Yaskawa INFORM job: DEMO_ROOF_UPPER_0625_3PAINT_66.JBI

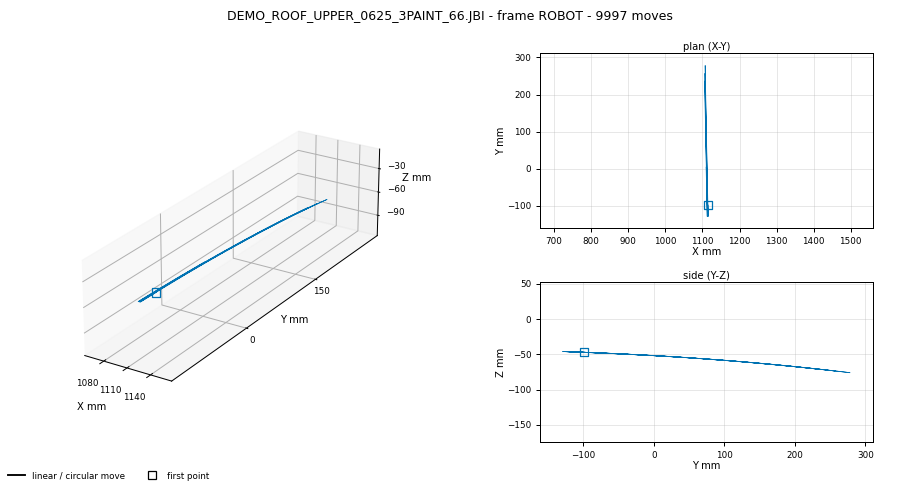
[picture p0: tool path of DEMO_ROOF_UPPER_0625_3PAINT_66.JBI in frame ROBOT, 9997 of 9997 moves have a stored position in this frame; points joined in program order, loops and branches not executed]
/JOB
//NAME DEMO_ROOF_UPPER_0625_3PAINT66
//POS
///NPOS 9997,0,0,0,0,0
///TOOL 0
///USER 0
///POSTYPE ROBOT
///RECTAN
///RCONF 1,0,0,0,0,0,0,0,0,0,0,0,0,0,0,0,0,0,0,0,0,0,0,0
C00000=1115.021,-98.188,-46.924,179.727,4.538,148.836
C00001=1115.026,-98.438,-46.914,179.727,4.533,148.835
C00002=1115.031,-98.688,-46.905,179.727,4.528,148.834
C00003=1115.036,-98.938,-46.894,179.727,4.523,148.833
C00004=1115.041,-99.188,-46.885,179.728,4.519,148.832
C00005=1115.047,-99.437,-46.875,179.728,4.513,148.830
C00006=1115.052,-99.653,-46.868,179.729,4.509,148.829
C00007=1115.056,-99.868,-46.859,179.728,4.505,148.828
C00008=1115.061,-100.083,-46.851,179.729,4.500,148.827
C00009=1115.066,-100.298,-46.842,179.729,4.496,148.826
C00010=1115.070,-100.513,-46.834,179.730,4.492,148.825
C00011=1115.075,-100.728,-46.826,179.729,4.488,148.824
C00012=1115.079,-100.943,-46.819,179.730,4.483,148.823
C00013=1115.084,-101.159,-46.811,179.731,4.479,148.822
C00014=1115.089,-101.408,-46.800,179.731,4.474,148.821
C00015=1115.094,-101.658,-46.791,179.731,4.469,148.820
C00016=1115.100,-101.908,-46.781,179.731,4.464,148.819
C00017=1115.105,-102.158,-46.772,179.732,4.459,148.817
C00018=1115.110,-102.407,-46.763,179.732,4.454,148.816
C00019=1115.116,-102.657,-46.753,179.733,4.449,148.815
C00020=1115.121,-102.907,-46.744,179.733,4.444,148.814
C00021=1115.127,-103.156,-46.734,179.733,4.439,148.813
C00022=1115.132,-103.406,-46.725,179.733,4.434,148.812
C00023=1115.137,-103.656,-46.716,179.734,4.429,148.810
C00024=1115.143,-103.906,-46.706,179.734,4.424,148.809
C00025=1115.148,-104.155,-46.697,179.735,4.419,148.808
C00026=1115.153,-104.405,-46.688,179.735,4.414,148.807
C00027=1115.159,-104.655,-46.678,179.735,4.409,148.806
C00028=1115.164,-104.905,-46.669,179.735,4.404,148.804
C00029=1115.170,-105.155,-46.660,179.736,4.399,148.803
C00030=1115.174,-105.404,-46.650,179.736,4.394,148.802
C00031=1115.180,-105.654,-46.641,179.737,4.389,148.801
C00032=1115.186,-105.904,-46.632,179.737,4.384,148.800
C00033=1115.190,-106.153,-46.622,179.737,4.379,148.798
C00034=1115.196,-106.403,-46.613,179.737,4.373,148.797
C00035=1115.201,-106.653,-46.604,179.738,4.369,148.796
C00036=1115.207,-106.903,-46.595,179.738,4.364,148.795
C00037=1115.211,-107.152,-46.585,179.739,4.359,148.794
C00038=1115.217,-107.402,-46.576,179.739,4.354,148.792
C00039=1115.223,-107.652,-46.567,179.739,4.348,148.791
C00040=1115.228,-107.902,-46.558,179.739,4.343,148.790
C00041=1115.233,-108.151,-46.548,179.739,4.338,148.789
C00042=1115.238,-108.402,-46.539,179.740,4.333,148.788
C00043=1115.244,-108.651,-46.530,179.741,4.329,148.786
C00044=1115.249,-108.901,-46.521,179.741,4.323,148.785
C00045=1115.254,-109.151,-46.512,179.741,4.318,148.784
C00046=1115.260,-109.401,-46.502,179.741,4.313,148.783
C00047=1115.265,-109.651,-46.493,179.742,4.308,148.782
C00048=1115.270,-109.900,-46.484,179.742,4.303,148.780
C00049=1115.275,-110.150,-46.475,179.742,4.298,148.779
C00050=1115.282,-110.400,-46.466,179.742,4.292,148.778
C00051=1115.287,-110.650,-46.457,179.743,4.287,148.777
C00052=1115.292,-110.899,-46.448,179.743,4.282,148.776
C00053=1115.297,-111.149,-46.439,179.743,4.277,148.774
C00054=1115.302,-111.399,-46.430,179.743,4.272,148.773
C00055=1115.308,-111.649,-46.420,179.744,4.267,148.772
C00056=1115.313,-111.899,-46.411,179.744,4.262,148.771
C00057=1115.318,-112.148,-46.402,179.745,4.257,148.770
C00058=1115.323,-112.398,-46.394,179.745,4.252,148.768
C00059=1115.329,-112.648,-46.385,179.745,4.247,148.767
C00060=1115.335,-112.898,-46.376,179.745,4.242,148.766
C00061=1115.340,-113.147,-46.367,179.746,4.236,148.764
C00062=1115.344,-113.363,-46.359,179.746,4.231,148.763
C00063=1115.349,-113.578,-46.350,179.746,4.227,148.763
C00064=1115.354,-113.793,-46.343,179.747,4.223,148.761
C00065=1115.359,-114.008,-46.335,179.747,4.218,148.760
C00066=1115.363,-114.223,-46.327,179.747,4.214,148.759
C00067=1115.367,-114.438,-46.320,179.747,4.209,148.758
C00068=1115.372,-114.654,-46.312,179.748,4.205,148.757
C00069=1115.376,-114.869,-46.305,179.748,4.200,148.756
C00070=1115.382,-115.118,-46.296,179.748,4.195,148.755
C00071=1115.388,-115.369,-46.286,179.749,4.190,148.754
C00072=1115.393,-115.619,-46.278,179.749,4.184,148.752
C00073=1115.398,-115.868,-46.269,179.749,4.179,148.751
C00074=1115.404,-116.118,-46.260,179.749,4.174,148.750
C00075=1115.409,-116.367,-46.251,179.750,4.169,148.749
C00076=1115.414,-116.617,-46.242,179.750,4.164,148.748
C00077=1115.419,-116.867,-46.233,179.751,4.158,148.746
C00078=1115.424,-117.117,-46.225,179.751,4.153,148.745
C00079=1115.430,-117.366,-46.216,179.751,4.148,148.744
C00080=1115.435,-117.616,-46.207,179.752,4.143,148.742
C00081=1115.441,-117.867,-46.198,179.752,4.137,148.741
C00082=1115.447,-118.117,-46.189,179.752,4.132,148.740
C00083=1115.452,-118.366,-46.181,179.752,4.127,148.739
C00084=1115.458,-118.616,-46.172,179.753,4.122,148.737
C00085=1115.463,-118.865,-46.163,179.753,4.116,148.736
C00086=1115.468,-119.115,-46.154,179.754,4.111,148.735
C00087=1115.473,-119.365,-46.145,179.754,4.106,148.734
C00088=1115.479,-119.614,-46.137,179.754,4.101,148.733
C00089=1115.484,-119.865,-46.129,179.755,4.096,148.731
C00090=1115.489,-120.115,-46.120,179.755,4.090,148.730
C00091=1115.495,-120.364,-46.111,179.755,4.084,148.729
C00092=1115.500,-120.614,-46.102,179.755,4.079,148.727
C00093=1115.506,-120.863,-46.093,179.756,4.074,148.726
C00094=1115.511,-121.113,-46.085,179.756,4.069,148.725
C00095=1115.516,-121.364,-46.076,179.757,4.063,148.724
C00096=1115.522,-121.613,-46.068,179.757,4.058,148.722
C00097=1115.527,-121.863,-46.059,179.757,4.053,148.721
C00098=1115.532,-122.113,-46.050,179.758,4.048,148.720
C00099=1115.538,-122.363,-46.042,179.758,4.042,148.718
C00100=1115.544,-122.612,-46.033,179.758,4.036,148.717
C00101=1115.549,-122.862,-46.024,179.758,4.031,148.716
C00102=1115.553,-123.112,-46.016,179.759,4.026,148.715
C00103=1115.559,-123.362,-46.008,179.760,4.020,148.713
C00104=1115.564,-123.611,-45.999,179.760,4.015,148.712
C00105=1115.570,-123.861,-45.990,179.760,4.010,148.711
C00106=1115.575,-124.111,-45.982,179.760,4.005,148.710
C00107=1115.581,-124.361,-45.974,179.761,3.998,148.708
C00108=1115.586,-124.611,-45.965,179.761,3.993,148.707
C00109=1115.591,-124.860,-45.956,179.761,3.988,148.706
C00110=1115.597,-125.110,-45.948,179.762,3.983,148.705
C00111=1115.602,-125.360,-45.939,179.762,3.977,148.703
C00112=1115.607,-125.610,-45.930,179.762,3.971,148.702
C00113=1115.613,-125.859,-45.923,179.762,3.966,148.701
C00114=1115.618,-126.109,-45.914,179.763,3.961,148.699
C00115=1115.623,-126.360,-45.906,179.763,3.955,148.698
C00116=1115.629,-126.609,-45.898,179.764,3.950,148.697
C00117=1115.634,-126.859,-45.889,179.764,3.944,148.695
C00118=1115.640,-127.074,-45.882,179.764,3.940,148.694
C00119=1115.644,-127.289,-45.875,179.765,3.935,148.693
C00120=1115.648,-127.504,-45.867,179.765,3.930,148.692
C00121=1115.654,-127.720,-45.860,179.765,3.926,148.691
C00122=1115.658,-127.935,-45.853,179.766,3.920,148.690
C00123=1115.662,-128.151,-45.845,179.765,3.916,148.689
C00124=1115.667,-128.366,-45.838,179.766,3.911,148.688
C00125=1115.671,-128.581,-45.831,179.767,3.906,148.686
C00126=1115.248,-128.571,-45.857,179.774,3.911,148.685
C00127=1115.243,-128.356,-45.864,179.774,3.916,148.686
C00128=1115.239,-128.141,-45.872,179.773,3.920,148.687
C00129=1115.234,-127.926,-45.878,179.773,3.925,148.689
C00130=1115.229,-127.710,-45.886,179.773,3.929,148.689
C00131=1115.225,-127.496,-45.893,179.772,3.934,148.691
C00132=1115.221,-127.280,-45.901,179.772,3.939,148.692
C00133=1115.216,-127.064,-45.908,179.772,3.943,148.693
C00134=1115.212,-126.849,-45.915,179.771,3.949,148.694
C00135=1115.206,-126.600,-45.923,179.771,3.954,148.695
C00136=1115.201,-126.350,-45.932,179.770,3.959,148.697
C00137=1115.195,-126.100,-45.941,179.770,3.965,148.698
C00138=1115.190,-125.851,-45.949,179.770,3.970,148.699
C00139=1115.184,-125.600,-45.957,179.769,3.976,148.701
C00140=1115.179,-125.350,-45.966,179.769,3.981,148.702
C00141=1115.173,-125.101,-45.975,179.769,3.986,148.703
C00142=1115.168,-124.851,-45.982,179.768,3.993,148.705
C00143=1115.163,-124.601,-45.991,179.768,3.998,148.706
C00144=1115.158,-124.351,-46.000,179.768,4.003,148.707
C00145=1115.152,-124.102,-46.008,179.768,4.008,148.708
C00146=1115.147,-123.852,-46.017,179.767,4.014,148.710
C00147=1115.142,-123.602,-46.026,179.766,4.019,148.711
C00148=1115.136,-123.353,-46.034,179.767,4.025,148.712
C00149=1115.130,-123.102,-46.042,179.766,4.030,148.713
C00150=1115.125,-122.853,-46.051,179.766,4.036,148.715
C00151=1115.120,-122.603,-46.060,179.765,4.041,148.716
C00152=1115.114,-122.354,-46.069,179.765,4.046,148.717
C00153=1115.109,-122.104,-46.078,179.765,4.051,148.718
C00154=1115.104,-121.853,-46.086,179.764,4.057,148.720
C00155=1115.099,-121.603,-46.095,179.764,4.062,148.721
C00156=1115.093,-121.354,-46.103,179.764,4.068,148.722
C00157=1115.088,-121.104,-46.112,179.764,4.073,148.724
C00158=1115.082,-120.854,-46.121,179.763,4.079,148.725
C00159=1115.077,-120.604,-46.129,179.763,4.084,148.726
C00160=1115.071,-120.355,-46.138,179.762,4.089,148.727
C00161=1115.066,-120.105,-46.147,179.762,4.094,148.729
C00162=1115.061,-119.855,-46.156,179.762,4.099,148.730
C00163=1115.056,-119.605,-46.164,179.761,4.105,148.731
C00164=1115.051,-119.355,-46.173,179.761,4.110,148.733
C00165=1115.045,-119.106,-46.182,179.760,4.115,148.734
C00166=1115.040,-118.856,-46.191,179.760,4.120,148.735
C00167=1115.034,-118.607,-46.200,179.760,4.125,148.736
C00168=1115.029,-118.356,-46.208,179.760,4.131,148.737
C00169=1115.024,-118.106,-46.217,179.759,4.136,148.739
C00170=1115.018,-117.857,-46.225,179.758,4.141,148.740
C00171=1115.013,-117.607,-46.234,179.759,4.147,148.741
C00172=1115.007,-117.357,-46.244,179.758,4.152,148.742
C00173=1115.002,-117.107,-46.253,179.758,4.158,148.744
C00174=1114.997,-116.857,-46.261,179.758,4.163,148.745
C00175=1114.991,-116.608,-46.270,179.757,4.168,148.746
C00176=1114.986,-116.358,-46.279,179.757,4.173,148.748
C00177=1114.981,-116.109,-46.288,179.757,4.179,148.749
C00178=1114.975,-115.859,-46.297,179.756,4.184,148.750
C00179=1114.970,-115.609,-46.306,179.756,4.189,148.751
C00180=1114.965,-115.359,-46.314,179.756,4.194,148.752
C00181=1114.959,-115.109,-46.324,179.756,4.199,148.754
C00182=1114.953,-114.860,-46.333,179.755,4.204,148.755
C00183=1114.949,-114.644,-46.340,179.754,4.209,148.756
C00184=1114.944,-114.429,-46.348,179.755,4.214,148.757
C00185=1114.940,-114.214,-46.356,179.754,4.218,148.758
C00186=1114.935,-113.999,-46.363,179.754,4.222,148.759
C00187=1114.931,-113.784,-46.371,179.754,4.227,148.760
C00188=1114.927,-113.569,-46.379,179.753,4.231,148.761
C00189=1114.922,-113.354,-46.387,179.753,4.236,148.762
C00190=1114.917,-113.138,-46.394,179.753,4.240,148.763
C00191=1114.911,-112.888,-46.404,179.752,4.245,148.765
C00192=1114.906,-112.638,-46.413,179.752,4.251,148.766
C00193=1114.901,-112.389,-46.422,179.752,4.256,148.767
C00194=1114.896,-112.139,-46.430,179.751,4.261,148.768
C00195=1114.891,-111.889,-46.439,179.751,4.266,148.769
C00196=1114.885,-111.639,-46.450,179.751,4.271,148.771
C00197=1114.879,-111.390,-46.458,179.751,4.276,148.772
C00198=1114.874,-111.140,-46.467,179.750,4.282,148.773
C00199=1114.869,-110.891,-46.476,179.749,4.286,148.774
C00200=1114.863,-110.640,-46.485,179.749,4.291,148.776
C00201=1114.858,-110.391,-46.494,179.749,4.296,148.777
C00202=1114.853,-110.141,-46.504,179.749,4.301,148.778
C00203=1114.848,-109.891,-46.513,179.748,4.307,148.779
C00204=1114.842,-109.641,-46.522,179.748,4.312,148.780
C00205=1114.837,-109.391,-46.531,179.748,4.317,148.782
C00206=1114.831,-109.142,-46.540,179.748,4.322,148.783
C00207=1114.827,-108.892,-46.550,179.747,4.327,148.784
C00208=1114.821,-108.642,-46.559,179.747,4.332,148.785
C00209=1114.816,-108.392,-46.568,179.746,4.337,148.786
C00210=1114.810,-108.142,-46.577,179.746,4.342,148.788
C00211=1114.804,-107.892,-46.586,179.746,4.347,148.789
C00212=1114.800,-107.643,-46.596,179.746,4.352,148.790
C00213=1114.794,-107.393,-46.605,179.745,4.357,148.791
C00214=1114.789,-107.143,-46.614,179.745,4.362,148.792
C00215=1114.784,-106.894,-46.624,179.745,4.368,148.794
C00216=1114.779,-106.644,-46.633,179.745,4.373,148.795
C00217=1114.773,-106.394,-46.642,179.743,4.378,148.796
C00218=1114.767,-106.144,-46.651,179.743,4.383,148.797
C00219=1114.763,-105.895,-46.661,179.743,4.388,148.799
C00220=1114.757,-105.645,-46.670,179.743,4.393,148.800
C00221=1114.752,-105.395,-46.679,179.742,4.398,148.801
C00222=1114.747,-105.145,-46.689,179.743,4.403,148.802
C00223=1114.741,-104.895,-46.698,179.742,4.408,148.803
C00224=1114.736,-104.645,-46.707,179.742,4.412,148.804
C00225=1114.731,-104.396,-46.717,179.741,4.418,148.805
C00226=1114.725,-104.146,-46.727,179.741,4.423,148.807
C00227=1114.720,-103.896,-46.735,179.741,4.428,148.808
C00228=1114.715,-103.647,-46.745,179.741,4.433,148.809
C00229=1114.709,-103.397,-46.755,179.740,4.437,148.810
C00230=1114.704,-103.148,-46.764,179.740,4.443,148.811
C00231=1114.698,-102.897,-46.774,179.739,4.448,148.813
C00232=1114.693,-102.648,-46.783,179.739,4.453,148.814
C00233=1114.688,-102.398,-46.792,179.739,4.458,148.815
C00234=1114.682,-102.148,-46.802,179.739,4.463,148.816
C00235=1114.677,-101.899,-46.811,179.738,4.468,148.817
C00236=1114.671,-101.649,-46.821,179.738,4.473,148.819
C00237=1114.667,-101.400,-46.830,179.737,4.478,148.820
C00238=1114.661,-101.149,-46.840,179.737,4.483,148.821
C00239=1114.657,-100.934,-46.849,179.737,4.487,148.822
C00240=1114.652,-100.719,-46.856,179.736,4.491,148.823
C00241=1114.647,-100.505,-46.864,179.736,4.495,148.824
C00242=1114.643,-100.289,-46.872,179.736,4.500,148.825
C00243=1114.638,-100.074,-46.881,179.735,4.504,148.826
C00244=1114.634,-99.858,-46.889,179.735,4.508,148.827
C00245=1114.629,-99.644,-46.898,179.735,4.512,148.828
C00246=1114.624,-99.429,-46.905,179.735,4.517,148.829
C00247=1114.619,-99.179,-46.916,179.735,4.522,148.830
C00248=1114.614,-98.929,-46.924,179.734,4.527,148.832
C00249=1114.609,-98.679,-46.935,179.734,4.532,148.833
C00250=1114.604,-98.429,-46.944,179.734,4.537,148.834
C00251=1114.598,-98.180,-46.954,179.733,4.542,148.835
C00252=1114.593,-97.930,-46.963,179.733,4.547,148.836
C00253=1114.587,-97.680,-46.973,179.732,4.552,148.837
C00254=1114.582,-97.431,-46.983,179.732,4.557,148.839
C00255=1114.576,-97.181,-46.992,179.732,4.562,148.840
C00256=1114.572,-96.932,-47.002,179.731,4.566,148.841
C00257=1114.566,-96.681,-47.012,179.731,4.571,148.842
C00258=1114.561,-96.431,-47.022,179.731,4.577,148.843
C00259=1114.555,-96.181,-47.031,179.730,4.582,148.845
C00260=1114.550,-95.932,-47.041,179.730,4.586,148.846
C00261=1114.545,-95.683,-47.051,179.729,4.591,148.847
C00262=1114.539,-95.432,-47.060,179.729,4.596,148.848
C00263=1114.534,-95.183,-47.070,179.728,4.601,148.849
C00264=1114.529,-94.933,-47.080,179.728,4.606,148.851
C00265=1114.523,-94.683,-47.090,179.728,4.611,148.852
C00266=1114.518,-94.434,-47.099,179.728,4.616,148.853
C00267=1114.513,-94.184,-47.110,179.727,4.621,148.854
C00268=1114.508,-93.934,-47.119,179.727,4.626,148.855
C00269=1114.502,-93.685,-47.129,179.726,4.630,148.857
C00270=1114.497,-93.434,-47.139,179.726,4.635,148.858
C00271=1114.492,-93.185,-47.148,179.725,4.640,148.859
C00272=1114.486,-92.935,-47.158,179.725,4.645,148.860
C00273=1114.481,-92.685,-47.169,179.724,4.649,148.861
C00274=1114.476,-92.436,-47.178,179.723,4.655,148.863
C00275=1114.471,-92.185,-47.188,179.723,4.659,148.864
C00276=1114.466,-91.936,-47.198,179.722,4.664,148.865
C00277=1114.460,-91.687,-47.208,179.722,4.669,148.866
C00278=1114.454,-91.436,-47.217,179.721,4.674,148.867
C00279=1114.449,-91.187,-47.227,179.721,4.679,148.869
C00280=1114.444,-90.937,-47.238,179.720,4.684,148.870
C00281=1114.439,-90.687,-47.248,179.720,4.689,148.871
C00282=1114.434,-90.438,-47.257,179.719,4.693,148.872
C00283=1114.428,-90.188,-47.267,179.719,4.698,148.874
C00284=1114.423,-89.938,-47.278,179.719,4.703,148.875
C00285=1114.418,-89.689,-47.287,179.718,4.708,148.876
C00286=1114.412,-89.438,-47.297,179.718,4.713,148.877
C00287=1114.407,-89.189,-47.307,179.717,4.718,148.879
C00288=1114.402,-88.939,-47.317,179.716,4.723,148.880
C00289=1114.397,-88.689,-47.327,179.716,4.728,148.881
C00290=1114.391,-88.440,-47.337,179.716,4.733,148.882
C00291=1114.386,-88.190,-47.347,179.715,4.737,148.883
C00292=1114.381,-87.940,-47.357,179.715,4.743,148.885
C00293=1114.375,-87.690,-47.367,179.714,4.748,148.886
C00294=1114.370,-87.441,-47.377,179.714,4.753,148.887
C00295=1114.366,-87.225,-47.386,179.714,4.757,148.888
C00296=1114.361,-87.011,-47.395,179.713,4.762,148.889
C00297=1114.357,-86.796,-47.403,179.713,4.766,148.890
C00298=1114.352,-86.581,-47.412,179.712,4.769,148.891
C00299=1114.348,-86.366,-47.421,179.712,4.775,148.892
C00300=1114.343,-86.150,-47.429,179.712,4.779,148.893
C00301=1114.338,-85.935,-47.438,179.711,4.783,148.894
C00302=1114.334,-85.720,-47.446,179.711,4.787,148.895
C00303=1114.328,-85.471,-47.457,179.711,4.792,148.897
C00304=1114.323,-85.221,-47.467,179.711,4.797,148.898
C00305=1114.318,-84.971,-47.477,179.710,4.802,148.899
C00306=1114.313,-84.722,-47.487,179.710,4.808,148.900
C00307=1114.308,-84.472,-47.497,179.710,4.813,148.902
C00308=1114.302,-84.222,-47.508,179.709,4.817,148.903
C00309=1114.296,-83.973,-47.518,179.709,4.823,148.904
C00310=1114.292,-83.723,-47.528,179.708,4.828,148.905
C00311=1114.287,-83.473,-47.538,179.708,4.833,148.906
C00312=1114.281,-83.224,-47.548,179.708,4.838,148.907
C00313=1114.276,-82.973,-47.559,179.708,4.843,148.909
C00314=1114.270,-82.724,-47.569,179.708,4.848,148.910
C00315=1114.265,-82.474,-47.579,179.706,4.853,148.911
C00316=1114.260,-82.224,-47.589,179.706,4.858,148.912
C00317=1114.255,-81.975,-47.599,179.706,4.863,148.914
C00318=1114.249,-81.725,-47.610,179.706,4.868,148.915
C00319=1114.244,-81.475,-47.620,179.706,4.874,148.916
C00320=1114.239,-81.225,-47.630,179.706,4.879,148.917
C00321=1114.233,-80.976,-47.641,179.705,4.884,148.918
C00322=1114.228,-80.726,-47.651,179.705,4.889,148.919
C00323=1114.223,-80.476,-47.661,179.705,4.894,148.921
C00324=1114.217,-80.227,-47.672,179.705,4.899,148.922
C00325=1114.213,-79.977,-47.682,179.705,4.905,148.923
C00326=1114.207,-79.727,-47.692,179.705,4.910,148.924
C00327=1114.202,-79.477,-47.702,179.704,4.915,148.925
C00328=1114.196,-79.227,-47.713,179.704,4.920,148.926
C00329=1114.191,-78.978,-47.724,179.704,4.925,148.928
C00330=1114.186,-78.728,-47.734,179.704,4.930,148.929
C00331=1114.181,-78.479,-47.744,179.704,4.935,148.930
C00332=1114.176,-78.228,-47.755,179.704,4.941,148.931
C00333=1114.170,-77.979,-47.765,179.704,4.946,148.932
C00334=1114.164,-77.729,-47.775,179.703,4.951,148.933
C00335=1114.159,-77.479,-47.786,179.703,4.956,148.935
C00336=1114.154,-77.230,-47.797,179.703,4.961,148.936
C00337=1114.149,-76.980,-47.807,179.703,4.966,148.937
C00338=1114.143,-76.730,-47.818,179.703,4.971,148.938
C00339=1114.138,-76.481,-47.828,179.703,4.977,148.939
C00340=1114.133,-76.231,-47.838,179.702,4.982,148.940
C00341=1114.128,-75.982,-47.849,179.702,4.987,148.942
C00342=1114.123,-75.731,-47.860,179.702,4.992,148.943
C00343=1114.117,-75.482,-47.870,179.702,4.997,148.944
C00344=1114.112,-75.232,-47.881,179.702,5.002,148.945
C00345=1114.107,-74.983,-47.892,179.702,5.007,148.946
C00346=1114.102,-74.732,-47.902,179.702,5.013,148.947
C00347=1114.096,-74.483,-47.912,179.702,5.019,148.949
C00348=1114.091,-74.233,-47.923,179.702,5.023,148.950
C00349=1114.086,-73.984,-47.934,179.702,5.028,148.951
C00350=1114.080,-73.734,-47.944,179.702,5.034,148.952
C00351=1114.076,-73.519,-47.953,179.702,5.038,148.953
C00352=1114.071,-73.304,-47.963,179.702,5.042,148.954
C00353=1114.067,-73.089,-47.972,179.702,5.047,148.955
C00354=1114.062,-72.874,-47.981,179.702,5.051,148.956
C00355=1114.058,-72.659,-47.991,179.702,5.056,148.957
C00356=1114.053,-72.444,-47.999,179.702,5.060,148.958
C00357=1114.049,-72.229,-48.009,179.702,5.065,148.959
C00358=1114.044,-72.015,-48.018,179.703,5.070,148.960
C00359=1114.039,-71.765,-48.029,179.703,5.075,148.961
C00360=1114.033,-71.515,-48.039,179.702,5.080,148.962
C00361=1114.028,-71.265,-48.050,179.702,5.085,148.963
C00362=1114.023,-71.015,-48.061,179.703,5.090,148.964
C00363=1114.018,-70.766,-48.071,179.703,5.095,148.965
C00364=1114.013,-70.516,-48.082,179.703,5.101,148.966
C00365=1114.007,-70.266,-48.093,179.703,5.106,148.967
C00366=1114.002,-70.017,-48.105,179.703,5.111,148.968
C00367=1113.996,-69.767,-48.115,179.703,5.116,148.970
C00368=1113.992,-69.517,-48.126,179.703,5.121,148.971
C00369=1113.986,-69.268,-48.136,179.704,5.127,148.972
C00370=1113.981,-69.018,-48.148,179.704,5.132,148.973
C00371=1113.976,-68.768,-48.159,179.704,5.137,148.974
C00372=1113.970,-68.519,-48.170,179.704,5.142,148.975
C00373=1113.965,-68.268,-48.180,179.704,5.147,148.976
C00374=1113.960,-68.020,-48.191,179.705,5.152,148.977
C00375=1113.955,-67.769,-48.202,179.705,5.158,148.978
C00376=1113.949,-67.520,-48.213,179.705,5.162,148.979
C00377=1113.944,-67.270,-48.224,179.705,5.168,148.980
C00378=1113.939,-67.020,-48.235,179.705,5.173,148.981
C00379=1113.934,-66.771,-48.245,179.706,5.178,148.982
C00380=1113.928,-66.521,-48.257,179.706,5.183,148.984
C00381=1113.923,-66.270,-48.268,179.706,5.188,148.984
C00382=1113.918,-66.022,-48.279,179.707,5.194,148.986
C00383=1113.913,-65.771,-48.289,179.707,5.199,148.987
C00384=1113.907,-65.522,-48.301,179.707,5.204,148.988
C00385=1113.902,-65.272,-48.312,179.707,5.209,148.989
C00386=1113.897,-65.022,-48.323,179.708,5.214,148.990
C00387=1113.891,-64.773,-48.334,179.708,5.219,148.991
C00388=1113.887,-64.523,-48.345,179.708,5.224,148.992
C00389=1113.882,-64.273,-48.356,179.709,5.230,148.993
C00390=1113.876,-64.024,-48.367,179.709,5.235,148.994
C00391=1113.871,-63.774,-48.379,179.710,5.240,148.995
C00392=1113.866,-63.524,-48.389,179.710,5.246,148.996
C00393=1113.861,-63.275,-48.400,179.711,5.250,148.997
C00394=1113.855,-63.025,-48.412,179.711,5.255,148.998
C00395=1113.850,-62.775,-48.423,179.711,5.260,148.999
C00396=1113.845,-62.526,-48.434,179.712,5.266,149.000
C00397=1113.840,-62.276,-48.446,179.712,5.271,149.001
C00398=1113.835,-62.026,-48.457,179.713,5.275,149.002
C00399=1113.829,-61.776,-48.468,179.713,5.281,149.003
C00400=1113.824,-61.527,-48.479,179.713,5.286,149.004
C00401=1113.819,-61.277,-48.490,179.714,5.291,149.005
C00402=1113.814,-61.027,-48.502,179.715,5.296,149.005
C00403=1113.808,-60.778,-48.512,179.715,5.301,149.006
C00404=1113.803,-60.528,-48.524,179.715,5.306,149.008
C00405=1113.798,-60.278,-48.536,179.716,5.312,149.008
C00406=1113.793,-60.029,-48.547,179.716,5.317,149.009
C00407=1113.788,-59.816,-48.557,179.716,5.320,149.010
C00408=1113.784,-59.603,-48.566,179.716,5.324,149.011
C00409=1113.780,-59.390,-48.576,179.716,5.328,149.012
C00410=1113.775,-59.178,-48.585,179.716,5.332,149.013
C00411=1113.770,-58.944,-48.596,179.716,5.337,149.014
C00412=1113.766,-58.711,-48.607,179.716,5.341,149.015
C00413=1113.760,-58.478,-48.617,179.716,5.345,149.016
C00414=1113.756,-58.245,-48.628,179.716,5.350,149.017
C00415=1113.751,-58.011,-48.639,179.715,5.354,149.018
C00416=1113.745,-57.778,-48.649,179.716,5.359,149.019
C00417=1113.741,-57.545,-48.660,179.715,5.363,149.020
C00418=1113.736,-57.311,-48.671,179.715,5.367,149.021
C00419=1113.731,-57.062,-48.682,179.715,5.372,149.022
C00420=1113.726,-56.812,-48.694,179.715,5.377,149.023
C00421=1113.721,-56.562,-48.705,179.714,5.381,149.024
C00422=1113.715,-56.313,-48.717,179.715,5.386,149.025
C00423=1113.710,-56.063,-48.728,179.714,5.390,149.026
C00424=1113.705,-55.813,-48.740,179.714,5.396,149.027
C00425=1113.700,-55.564,-48.751,179.715,5.400,149.028
C00426=1113.695,-55.314,-48.763,179.714,5.405,149.029
C00427=1113.690,-55.064,-48.774,179.714,5.410,149.031
C00428=1113.684,-54.815,-48.786,179.714,5.414,149.032
C00429=1113.679,-54.565,-48.797,179.713,5.419,149.033
C00430=1113.674,-54.315,-48.809,179.713,5.424,149.034
C00431=1113.669,-54.066,-48.821,179.713,5.428,149.035
C00432=1113.664,-53.816,-48.832,179.713,5.433,149.036
C00433=1113.658,-53.566,-48.844,179.713,5.438,149.037
C00434=1113.653,-53.317,-48.855,179.713,5.442,149.038
C00435=1113.648,-53.067,-48.867,179.713,5.447,149.039
C00436=1113.643,-52.817,-48.878,179.712,5.452,149.040
C00437=1113.638,-52.568,-48.890,179.712,5.456,149.041
C00438=1113.632,-52.318,-48.902,179.712,5.461,149.042
C00439=1113.627,-52.068,-48.913,179.712,5.466,149.044
C00440=1113.622,-51.818,-48.925,179.712,5.471,149.044
C00441=1113.617,-51.569,-48.936,179.711,5.475,149.046
C00442=1113.611,-51.319,-48.948,179.711,5.480,149.047
C00443=1113.606,-51.069,-48.960,179.712,5.485,149.048
C00444=1113.601,-50.820,-48.971,179.711,5.489,149.049
C00445=1113.596,-50.570,-48.983,179.711,5.494,149.050
C00446=1113.590,-50.320,-48.995,179.711,5.499,149.051
C00447=1113.586,-50.071,-49.007,179.711,5.503,149.052
C00448=1113.581,-49.821,-49.019,179.711,5.508,149.053
C00449=1113.574,-49.572,-49.030,179.711,5.512,149.054
C00450=1113.570,-49.322,-49.042,179.710,5.518,149.055
C00451=1113.564,-49.072,-49.053,179.710,5.523,149.056
C00452=1113.559,-48.822,-49.065,179.710,5.527,149.058
C00453=1113.554,-48.572,-49.077,179.710,5.532,149.058
C00454=1113.549,-48.323,-49.089,179.709,5.536,149.060
C00455=1113.544,-48.073,-49.101,179.709,5.541,149.061
C00456=1113.539,-47.824,-49.112,179.710,5.546,149.062
C00457=1113.534,-47.574,-49.124,179.709,5.550,149.063
C00458=1113.528,-47.324,-49.136,179.709,5.555,149.064
C00459=1113.524,-47.075,-49.148,179.709,5.561,149.065
C00460=1113.518,-46.825,-49.160,179.709,5.564,149.066
C00461=1113.512,-46.576,-49.172,179.709,5.570,149.067
C00462=1113.507,-46.326,-49.183,179.708,5.574,149.068
C00463=1113.503,-46.111,-49.194,179.708,5.578,149.069
C00464=1113.498,-45.896,-49.204,179.708,5.583,149.070
C00465=1113.494,-45.682,-49.214,179.708,5.587,149.071
C00466=1113.490,-45.467,-49.224,179.708,5.591,149.072
C00467=1113.485,-45.252,-49.235,179.708,5.594,149.073
C00468=1113.481,-45.037,-49.246,179.708,5.598,149.074
C00469=1113.476,-44.822,-49.256,179.707,5.602,149.075
C00470=1113.472,-44.608,-49.266,179.707,5.606,149.076
C00471=1113.467,-44.358,-49.277,179.707,5.611,149.077
C00472=1113.461,-44.108,-49.290,179.707,5.616,149.078
C00473=1113.456,-43.858,-49.302,179.707,5.620,149.079
C00474=1113.451,-43.609,-49.313,179.707,5.626,149.080
C00475=1113.446,-43.359,-49.326,179.706,5.630,149.081
C00476=1113.441,-43.110,-49.338,179.706,5.635,149.082
C00477=1113.435,-42.860,-49.350,179.707,5.640,149.083
C00478=1113.430,-42.610,-49.362,179.707,5.645,149.084
C00479=1113.426,-42.361,-49.373,179.708,5.650,149.085
C00480=1113.420,-42.111,-49.385,179.709,5.656,149.086
C00481=1113.415,-41.861,-49.398,179.710,5.660,149.087
C00482=1113.410,-41.611,-49.410,179.711,5.666,149.088
C00483=1113.404,-41.362,-49.422,179.712,5.671,149.089
C00484=1113.399,-41.112,-49.434,179.712,5.676,149.090
C00485=1113.394,-40.863,-49.446,179.714,5.681,149.090
C00486=1113.389,-40.613,-49.458,179.714,5.686,149.091
C00487=1113.384,-40.363,-49.470,179.715,5.692,149.092
C00488=1113.379,-40.114,-49.483,179.716,5.696,149.093
C00489=1113.373,-39.864,-49.495,179.716,5.701,149.094
C00490=1113.368,-39.615,-49.507,179.718,5.706,149.095
C00491=1113.363,-39.365,-49.519,179.718,5.711,149.095
C00492=1113.358,-39.116,-49.532,179.718,5.716,149.096
C00493=1113.352,-38.866,-49.544,179.719,5.721,149.097
C00494=1113.347,-38.616,-49.556,179.720,5.726,149.098
C00495=1113.342,-38.366,-49.568,179.721,5.730,149.099
C00496=1113.337,-38.116,-49.581,179.721,5.735,149.100
C00497=1113.332,-37.866,-49.593,179.722,5.740,149.101
C00498=1113.327,-37.617,-49.605,179.723,5.745,149.102
C00499=1113.322,-37.368,-49.617,179.724,5.750,149.102
C00500=1113.317,-37.118,-49.629,179.724,5.755,149.103
C00501=1113.312,-36.869,-49.642,179.725,5.759,149.104
C00502=1113.306,-36.619,-49.654,179.725,5.764,149.105
C00503=1113.301,-36.370,-49.666,179.726,5.768,149.106
C00504=1113.296,-36.120,-49.679,179.726,5.773,149.107
C00505=1113.291,-35.870,-49.691,179.727,5.778,149.107
C00506=1113.286,-35.620,-49.704,179.727,5.783,149.108
C00507=1113.281,-35.371,-49.717,179.728,5.787,149.109
C00508=1113.275,-35.121,-49.729,179.728,5.791,149.110
C00509=1113.270,-34.871,-49.742,179.729,5.796,149.111
C00510=1113.264,-34.622,-49.754,179.729,5.800,149.112
C00511=1113.259,-34.372,-49.766,179.729,5.805,149.113
C00512=1113.254,-34.122,-49.779,179.730,5.810,149.114
C00513=1113.249,-33.873,-49.792,179.731,5.814,149.114
C00514=1113.244,-33.623,-49.804,179.731,5.818,149.115
C00515=1113.239,-33.374,-49.816,179.731,5.823,149.116
C00516=1113.234,-33.124,-49.829,179.732,5.828,149.117
C00517=1113.229,-32.875,-49.841,179.732,5.832,149.118
C00518=1113.224,-32.624,-49.854,179.732,5.836,149.119
C00519=1113.219,-32.410,-49.865,179.732,5.840,149.119
C00520=1113.215,-32.195,-49.876,179.732,5.844,149.120
C00521=1113.210,-31.980,-49.886,179.733,5.847,149.121
C00522=1113.206,-31.766,-49.897,179.733,5.851,149.122
C00523=1113.201,-31.551,-49.908,179.733,5.856,149.123
C00524=1113.197,-31.337,-49.918,179.734,5.859,149.123
C00525=1113.192,-31.122,-49.930,179.734,5.863,149.124
C00526=1113.188,-30.907,-49.941,179.734,5.867,149.125
C00527=1113.183,-30.658,-49.953,179.734,5.871,149.126
C00528=1113.178,-30.408,-49.966,179.734,5.875,149.127
C00529=1113.173,-30.159,-49.978,179.734,5.879,149.128
C00530=1113.167,-29.909,-49.991,179.734,5.884,149.129
C00531=1113.162,-29.659,-50.004,179.734,5.888,149.130
C00532=1113.157,-29.410,-50.017,179.734,5.892,149.131
C00533=1113.152,-29.160,-50.029,179.734,5.897,149.131
C00534=1113.147,-28.911,-50.042,179.734,5.901,149.132
C00535=1113.143,-28.661,-50.055,179.734,5.906,149.133
C00536=1113.136,-28.411,-50.067,179.734,5.910,149.134
C00537=1113.131,-28.161,-50.080,179.734,5.914,149.135
C00538=1113.126,-27.912,-50.092,179.734,5.919,149.136
C00539=1113.122,-27.662,-50.105,179.734,5.923,149.137
C00540=1113.116,-27.413,-50.118,179.733,5.927,149.138
C00541=1113.111,-27.163,-50.131,179.733,5.931,149.139
C00542=1113.106,-26.913,-50.144,179.733,5.936,149.140
C00543=1113.101,-26.664,-50.157,179.733,5.940,149.141
C00544=1113.096,-26.414,-50.169,179.733,5.944,149.142
C00545=1113.091,-26.165,-50.182,179.732,5.949,149.143
C00546=1113.085,-25.915,-50.195,179.732,5.954,149.145
C00547=1113.080,-25.665,-50.208,179.732,5.958,149.145
C00548=1113.075,-25.416,-50.221,179.732,5.962,149.146
C00549=1113.071,-25.166,-50.234,179.733,5.967,149.147
C00550=1113.065,-24.916,-50.247,179.733,5.972,149.148
C00551=1113.060,-24.667,-50.259,179.734,5.977,149.149
C00552=1113.055,-24.418,-50.272,179.734,5.981,149.150
C00553=1113.050,-24.168,-50.285,179.735,5.986,149.151
C00554=1113.044,-23.918,-50.298,179.735,5.991,149.152
C00555=1113.039,-23.669,-50.311,179.736,5.995,149.153
C00556=1113.035,-23.419,-50.324,179.737,6.001,149.154
C00557=1113.029,-23.169,-50.337,179.737,6.006,149.154
C00558=1113.024,-22.920,-50.350,179.738,6.010,149.155
C00559=1113.019,-22.670,-50.363,179.738,6.015,149.156
C00560=1113.013,-22.420,-50.376,179.739,6.020,149.157
C00561=1113.008,-22.171,-50.388,179.739,6.025,149.158
C00562=1113.003,-21.921,-50.401,179.740,6.029,149.159
C00563=1112.998,-21.671,-50.414,179.740,6.034,149.160
C00564=1112.993,-21.422,-50.427,179.741,6.039,149.161
C00565=1112.988,-21.172,-50.440,179.741,6.044,149.162
C00566=1112.982,-20.923,-50.454,179.741,6.048,149.163
C00567=1112.978,-20.673,-50.467,179.742,6.053,149.163
C00568=1112.972,-20.423,-50.480,179.742,6.057,149.164
C00569=1112.967,-20.174,-50.493,179.742,6.062,149.165
C00570=1112.962,-19.924,-50.506,179.743,6.066,149.166
C00571=1112.957,-19.674,-50.519,179.743,6.071,149.167
C00572=1112.952,-19.425,-50.533,179.744,6.076,149.168
C00573=1112.946,-19.175,-50.546,179.744,6.081,149.169
C00574=1112.941,-18.926,-50.558,179.745,6.085,149.170
C00575=1112.937,-18.711,-50.570,179.746,6.090,149.170
C00576=1112.933,-18.497,-50.581,179.746,6.093,149.171
C00577=1112.928,-18.282,-50.592,179.747,6.098,149.172
C00578=1112.924,-18.067,-50.603,179.747,6.101,149.173
C00579=1112.920,-17.853,-50.616,179.747,6.105,149.173
C00580=1112.916,-17.639,-50.627,179.748,6.110,149.174
C00581=1112.911,-17.424,-50.638,179.748,6.113,149.175
C00582=1112.906,-17.209,-50.649,179.749,6.118,149.176
C00583=1112.901,-16.959,-50.663,179.750,6.122,149.176
C00584=1112.896,-16.710,-50.676,179.750,6.126,149.177
C00585=1112.892,-16.460,-50.689,179.750,6.131,149.178
C00586=1112.886,-16.211,-50.702,179.751,6.136,149.179
C00587=1112.881,-15.961,-50.716,179.751,6.140,149.180
C00588=1112.876,-15.712,-50.729,179.752,6.145,149.181
C00589=1112.871,-15.462,-50.742,179.752,6.150,149.182
C00590=1112.866,-15.213,-50.756,179.753,6.154,149.183
C00591=1112.861,-14.963,-50.769,179.753,6.159,149.183
C00592=1112.855,-14.713,-50.782,179.754,6.163,149.184
C00593=1112.850,-14.463,-50.796,179.755,6.168,149.185
C00594=1112.845,-14.214,-50.809,179.755,6.173,149.186
C00595=1112.840,-13.964,-50.823,179.756,6.178,149.187
C00596=1112.835,-13.715,-50.836,179.756,6.182,149.188
C00597=1112.830,-13.465,-50.849,179.757,6.187,149.188
C00598=1112.825,-13.216,-50.863,179.758,6.191,149.189
C00599=1112.820,-12.966,-50.876,179.758,6.195,149.190
C00600=1112.815,-12.717,-50.890,179.758,6.200,149.191
C00601=1112.810,-12.467,-50.903,179.759,6.204,149.192
C00602=1112.804,-12.218,-50.917,179.760,6.209,149.193
C00603=1112.800,-11.968,-50.930,179.760,6.214,149.193
C00604=1112.794,-11.719,-50.944,179.761,6.218,149.194
C00605=1112.789,-11.469,-50.957,179.762,6.223,149.195
C00606=1112.784,-11.220,-50.971,179.762,6.228,149.196
C00607=1112.779,-10.969,-50.984,179.763,6.232,149.197
C00608=1112.774,-10.721,-50.998,179.763,6.237,149.198
C00609=1112.769,-10.470,-51.011,179.764,6.241,149.198
C00610=1112.764,-10.220,-51.026,179.764,6.245,149.199
C00611=1112.758,-9.971,-51.038,179.765,6.250,149.200
C00612=1112.753,-9.721,-51.052,179.765,6.255,149.201
C00613=1112.748,-9.472,-51.066,179.766,6.259,149.202
C00614=1112.743,-9.222,-51.079,179.767,6.264,149.203
C00615=1112.738,-8.973,-51.094,179.767,6.268,149.204
C00616=1112.733,-8.723,-51.107,179.768,6.273,149.204
C00617=1112.728,-8.474,-51.120,179.769,6.278,149.205
C00618=1112.723,-8.224,-51.134,179.769,6.282,149.206
C00619=1112.718,-7.974,-51.148,179.770,6.287,149.207
C00620=1112.713,-7.725,-51.162,179.771,6.291,149.208
C00621=1112.707,-7.475,-51.175,179.771,6.295,149.208
C00622=1112.703,-7.226,-51.189,179.771,6.300,149.209
C00623=1112.697,-6.977,-51.203,179.772,6.305,149.210
C00624=1112.692,-6.727,-51.216,179.773,6.309,149.211
C00625=1112.687,-6.477,-51.230,179.773,6.314,149.212
C00626=1112.682,-6.228,-51.244,179.774,6.318,149.213
C00627=1112.677,-5.978,-51.258,179.775,6.323,149.213
C00628=1112.672,-5.728,-51.271,179.775,6.327,149.214
C00629=1112.667,-5.479,-51.285,179.776,6.332,149.215
C00630=1112.662,-5.229,-51.300,179.776,6.336,149.216
C00631=1112.657,-5.015,-51.311,179.777,6.340,149.217
C00632=1112.653,-4.800,-51.323,179.777,6.344,149.217
C00633=1112.649,-4.586,-51.335,179.778,6.348,149.218
C00634=1112.645,-4.371,-51.347,179.778,6.352,149.219
C00635=1112.640,-4.157,-51.359,179.779,6.355,149.219
C00636=1112.635,-3.943,-51.370,179.779,6.360,149.220
C00637=1112.632,-3.728,-51.383,179.780,6.364,149.221
C00638=1112.627,-3.513,-51.394,179.780,6.367,149.222
C00639=1112.622,-3.264,-51.408,179.781,6.372,149.222
C00640=1112.617,-3.014,-51.423,179.782,6.376,149.223
C00641=1112.611,-2.765,-51.437,179.782,6.381,149.224
C00642=1112.606,-2.515,-51.451,179.783,6.386,149.225
C00643=1112.601,-2.265,-51.465,179.783,6.390,149.226
C00644=1112.596,-2.016,-51.478,179.784,6.395,149.226
C00645=1112.591,-1.766,-51.492,179.785,6.399,149.227
C00646=1112.586,-1.517,-51.506,179.785,6.403,149.228
C00647=1112.581,-1.267,-51.521,179.786,6.408,149.229
C00648=1112.576,-1.018,-51.534,179.786,6.412,149.230
C00649=1112.571,-0.768,-51.549,179.787,6.417,149.231
C00650=1112.566,-0.519,-51.563,179.787,6.422,149.232
C00651=1112.561,-0.269,-51.577,179.788,6.426,149.232
C00652=1112.555,-0.020,-51.591,179.789,6.431,149.233
C00653=1112.551,0.230,-51.605,179.789,6.436,149.234
C00654=1112.546,0.480,-51.618,179.790,6.440,149.235
C00655=1112.541,0.730,-51.633,179.790,6.444,149.236
C00656=1112.535,0.979,-51.647,179.791,6.449,149.236
C00657=1112.531,1.228,-51.661,179.791,6.453,149.237
C00658=1112.526,1.478,-51.675,179.792,6.458,149.238
C00659=1112.521,1.728,-51.689,179.793,6.462,149.239
C00660=1112.515,1.977,-51.703,179.793,6.467,149.240
C00661=1112.510,2.226,-51.718,179.794,6.472,149.241
C00662=1112.505,2.476,-51.732,179.795,6.476,149.241
C00663=1112.500,2.726,-51.746,179.795,6.481,149.242
C00664=1112.495,2.976,-51.760,179.796,6.486,149.243
C00665=1112.490,3.224,-51.775,179.796,6.490,149.244
C00666=1112.485,3.474,-51.789,179.797,6.494,149.245
C00667=1112.480,3.723,-51.804,179.797,6.499,149.246
C00668=1112.475,3.973,-51.818,179.798,6.503,149.246
C00669=1112.470,4.223,-51.832,179.798,6.508,149.247
C00670=1112.465,4.472,-51.846,179.799,6.512,149.248
C00671=1112.460,4.721,-51.860,179.800,6.517,149.249
C00672=1112.455,4.971,-51.875,179.801,6.522,149.250
C00673=1112.450,5.221,-51.889,179.801,6.526,149.251
C00674=1112.445,5.471,-51.903,179.802,6.531,149.252
C00675=1112.439,5.720,-51.919,179.803,6.535,149.252
C00676=1112.434,5.970,-51.933,179.803,6.540,149.253
C00677=1112.429,6.219,-51.947,179.804,6.545,149.254
C00678=1112.424,6.468,-51.961,179.804,6.550,149.255
C00679=1112.419,6.718,-51.976,179.804,6.553,149.256
C00680=1112.414,6.968,-51.990,179.805,6.558,149.256
C00681=1112.409,7.217,-52.005,179.806,6.563,149.257
C00682=1112.404,7.467,-52.019,179.806,6.567,149.258
C00683=1112.399,7.716,-52.033,179.807,6.572,149.259
C00684=1112.395,7.966,-52.048,179.807,6.577,149.260
C00685=1112.389,8.215,-52.063,179.808,6.581,149.261
C00686=1112.384,8.465,-52.077,179.809,6.586,149.261
C00687=1112.380,8.679,-52.090,179.809,6.590,149.262
C00688=1112.376,8.894,-52.102,179.810,6.594,149.263
C00689=1112.371,9.108,-52.115,179.810,6.597,149.264
C00690=1112.367,9.323,-52.127,179.810,6.601,149.265
C00691=1112.362,9.537,-52.139,179.811,6.606,149.265
C00692=1112.358,9.752,-52.152,179.812,6.609,149.266
C00693=1112.353,9.965,-52.164,179.812,6.613,149.267
C00694=1112.349,10.180,-52.176,179.813,6.617,149.267
C00695=1112.344,10.430,-52.192,179.813,6.622,149.268
C00696=1112.339,10.679,-52.206,179.813,6.626,149.269
C00697=1112.334,10.929,-52.221,179.814,6.630,149.270
C00698=1112.329,11.178,-52.236,179.815,6.635,149.271
C00699=1112.324,11.428,-52.250,179.815,6.640,149.272
C00700=1112.319,11.677,-52.265,179.816,6.645,149.273
C00701=1112.314,11.927,-52.280,179.816,6.649,149.273
C00702=1112.309,12.177,-52.294,179.817,6.654,149.274
C00703=1112.305,12.426,-52.309,179.817,6.658,149.275
C00704=1112.299,12.676,-52.324,179.818,6.662,149.276
C00705=1112.294,12.925,-52.339,179.819,6.667,149.276
C00706=1112.289,13.174,-52.353,179.819,6.671,149.277
C00707=1112.284,13.424,-52.368,179.820,6.676,149.278
C00708=1112.279,13.674,-52.383,179.821,6.681,149.279
C00709=1112.274,13.923,-52.397,179.822,6.685,149.280
C00710=1112.269,14.172,-52.412,179.822,6.689,149.281
C00711=1112.264,14.422,-52.427,179.822,6.694,149.282
C00712=1112.259,14.671,-52.442,179.823,6.698,149.282
C00713=1112.254,14.921,-52.456,179.824,6.703,149.283
C00714=1112.249,15.171,-52.472,179.824,6.707,149.284
C00715=1112.244,15.420,-52.486,179.825,6.712,149.285
C00716=1112.239,15.669,-52.501,179.826,6.716,149.286
C00717=1112.233,15.919,-52.516,179.826,6.720,149.286
C00718=1112.229,16.169,-52.531,179.827,6.725,149.287
C00719=1112.224,16.418,-52.545,179.827,6.729,149.288
C00720=1112.218,16.668,-52.561,179.828,6.734,149.289
C00721=1112.214,16.917,-52.576,179.829,6.738,149.289
C00722=1112.209,17.166,-52.590,179.830,6.743,149.290
C00723=1112.203,17.416,-52.606,179.830,6.747,149.291
C00724=1112.198,17.666,-52.620,179.831,6.751,149.292
C00725=1112.193,17.915,-52.636,179.832,6.756,149.293
C00726=1112.188,18.164,-52.651,179.832,6.760,149.293
C00727=1112.183,18.414,-52.665,179.833,6.765,149.294
C00728=1112.178,18.663,-52.681,179.834,6.769,149.295
C00729=1112.173,18.913,-52.695,179.834,6.773,149.296
C00730=1112.168,19.162,-52.710,179.835,6.778,149.297
C00731=1112.164,19.412,-52.726,179.836,6.782,149.297
C00732=1112.158,19.662,-52.741,179.836,6.787,149.298
C00733=1112.153,19.911,-52.756,179.837,6.791,149.299
C00734=1112.149,20.160,-52.771,179.838,6.796,149.300
C00735=1112.143,20.410,-52.786,179.838,6.799,149.300
C00736=1112.138,20.659,-52.801,179.839,6.804,149.301
C00737=1112.133,20.909,-52.816,179.840,6.808,149.302
C00738=1112.128,21.158,-52.831,179.841,6.813,149.303
C00739=1112.123,21.408,-52.846,179.842,6.817,149.303
C00740=1112.119,21.658,-52.861,179.843,6.821,149.304
C00741=1112.113,21.907,-52.877,179.843,6.825,149.305
C00742=1112.108,22.156,-52.892,179.844,6.830,149.306
C00743=1112.104,22.371,-52.905,179.845,6.834,149.306
C00744=1112.099,22.585,-52.918,179.845,6.838,149.307
C00745=1112.095,22.799,-52.931,179.846,6.841,149.307
C00746=1112.091,23.014,-52.944,179.846,6.845,149.308
C00747=1112.087,23.228,-52.957,179.847,6.849,149.309
C00748=1112.082,23.442,-52.970,179.847,6.852,149.309
C00749=1112.078,23.656,-52.984,179.848,6.856,149.310
C00750=1112.074,23.871,-52.996,179.849,6.859,149.311
C00751=1112.069,24.120,-53.012,179.849,6.864,149.311
C00752=1112.064,24.369,-53.027,179.850,6.868,149.312
C00753=1112.059,24.619,-53.042,179.851,6.872,149.313
C00754=1112.054,24.869,-53.058,179.852,6.877,149.314
C00755=1112.049,25.118,-53.073,179.853,6.881,149.314
C00756=1112.043,25.368,-53.088,179.854,6.885,149.315
C00757=1112.039,25.617,-53.103,179.854,6.890,149.316
C00758=1112.033,25.867,-53.119,179.855,6.894,149.316
C00759=1112.029,26.117,-53.135,179.856,6.898,149.317
C00760=1112.024,26.366,-53.150,179.857,6.903,149.318
C00761=1112.019,26.615,-53.165,179.857,6.906,149.319
C00762=1112.013,26.865,-53.181,179.858,6.911,149.319
C00763=1112.008,27.114,-53.196,179.859,6.915,149.320
C00764=1112.004,27.364,-53.212,179.860,6.919,149.321
C00765=1111.999,27.613,-53.227,179.861,6.924,149.322
C00766=1111.994,27.862,-53.242,179.862,6.928,149.322
C00767=1111.988,28.112,-53.258,179.862,6.932,149.323
C00768=1111.984,28.361,-53.273,179.864,6.936,149.323
C00769=1111.979,28.611,-53.289,179.864,6.941,149.324
C00770=1111.973,28.860,-53.305,179.865,6.945,149.325
C00771=1111.968,29.110,-53.320,179.866,6.950,149.326
C00772=1111.964,29.359,-53.335,179.867,6.953,149.326
C00773=1111.959,29.609,-53.351,179.868,6.957,149.327
C00774=1111.953,29.858,-53.367,179.869,6.962,149.328
C00775=1111.949,30.108,-53.382,179.869,6.966,149.329
C00776=1111.944,30.357,-53.398,179.870,6.971,149.329
C00777=1111.938,30.607,-53.413,179.871,6.974,149.330
C00778=1111.933,30.856,-53.429,179.872,6.979,149.330
C00779=1111.929,31.105,-53.445,179.873,6.983,149.331
C00780=1111.924,31.355,-53.460,179.874,6.987,149.332
C00781=1111.919,31.604,-53.476,179.875,6.992,149.332
C00782=1111.914,31.854,-53.492,179.876,6.995,149.333
C00783=1111.909,32.103,-53.507,179.876,7.000,149.334
C00784=1111.904,32.353,-53.523,179.877,7.004,149.335
C00785=1111.899,32.602,-53.539,179.878,7.008,149.335
C00786=1111.894,32.852,-53.555,179.879,7.013,149.336
C00787=1111.889,33.101,-53.570,179.880,7.016,149.337
C00788=1111.884,33.351,-53.586,179.881,7.020,149.337
C00789=1111.879,33.600,-53.601,179.882,7.025,149.338
C00790=1111.874,33.849,-53.618,179.883,7.029,149.339
C00791=1111.869,34.099,-53.634,179.884,7.033,149.339
C00792=1111.864,34.349,-53.649,179.884,7.037,149.340
C00793=1111.859,34.598,-53.664,179.886,7.041,149.341
C00794=1111.855,34.847,-53.681,179.887,7.046,149.341
C00795=1111.849,35.097,-53.696,179.888,7.050,149.342
C00796=1111.844,35.346,-53.712,179.889,7.054,149.342
C00797=1111.839,35.596,-53.728,179.889,7.058,149.343
C00798=1111.834,35.845,-53.744,179.890,7.062,149.344
C00799=1111.830,36.059,-53.758,179.891,7.066,149.344
C00800=1111.825,36.273,-53.772,179.892,7.069,149.345
C00801=1111.821,36.488,-53.785,179.893,7.073,149.346
C00802=1111.817,36.702,-53.799,179.894,7.076,149.346
C00803=1111.813,36.916,-53.812,179.895,7.080,149.347
C00804=1111.809,37.130,-53.826,179.895,7.084,149.347
C00805=1111.805,37.345,-53.840,179.896,7.087,149.348
C00806=1111.800,37.559,-53.853,179.896,7.091,149.348
C00807=1111.795,37.809,-53.869,179.898,7.095,149.349
C00808=1111.790,38.057,-53.885,179.899,7.099,149.349
C00809=1111.785,38.307,-53.901,179.900,7.103,149.350
C00810=1111.780,38.556,-53.918,179.901,7.107,149.351
C00811=1111.775,38.806,-53.933,179.902,7.111,149.351
C00812=1111.770,39.056,-53.949,179.903,7.115,149.352
C00813=1111.765,39.305,-53.966,179.904,7.120,149.353
C00814=1111.760,39.555,-53.981,179.905,7.124,149.353
C00815=1111.756,39.804,-53.998,179.906,7.128,149.354
C00816=1111.750,40.053,-54.014,179.906,7.132,149.355
C00817=1111.745,40.302,-54.030,179.907,7.136,149.355
C00818=1111.740,40.552,-54.046,179.909,7.140,149.356
C00819=1111.735,40.801,-54.062,179.910,7.144,149.356
C00820=1111.730,41.051,-54.078,179.911,7.148,149.357
C00821=1111.725,41.300,-54.094,179.912,7.152,149.358
C00822=1111.721,41.550,-54.110,179.913,7.156,149.358
C00823=1111.715,41.799,-54.127,179.914,7.161,149.359
C00824=1111.711,42.049,-54.143,179.915,7.165,149.360
C00825=1111.706,42.298,-54.159,179.916,7.169,149.360
C00826=1111.701,42.547,-54.176,179.917,7.172,149.361
C00827=1111.696,42.797,-54.191,179.918,7.177,149.361
C00828=1111.691,43.046,-54.208,179.919,7.181,149.362
C00829=1111.685,43.296,-54.224,179.920,7.185,149.363
C00830=1111.681,43.545,-54.241,179.922,7.189,149.363
C00831=1111.676,43.794,-54.257,179.922,7.193,149.364
C00832=1111.671,44.044,-54.273,179.923,7.197,149.364
C00833=1111.666,44.294,-54.290,179.924,7.201,149.365
C00834=1111.661,44.543,-54.305,179.925,7.206,149.366
C00835=1111.656,44.793,-54.322,179.927,7.209,149.366
C00836=1111.651,45.041,-54.338,179.927,7.213,149.367
C00837=1111.647,45.292,-54.354,179.928,7.217,149.368
C00838=1111.641,45.541,-54.371,179.929,7.222,149.368
C00839=1111.636,45.790,-54.388,179.931,7.226,149.369
C00840=1111.631,46.039,-54.404,179.932,7.230,149.369
C00841=1111.626,46.289,-54.420,179.933,7.233,149.370
C00842=1111.622,46.538,-54.437,179.934,7.238,149.371
C00843=1111.617,46.787,-54.453,179.935,7.242,149.371
C00844=1111.612,47.037,-54.470,179.936,7.246,149.372
C00845=1111.606,47.286,-54.486,179.937,7.250,149.372
C00846=1111.602,47.536,-54.502,179.939,7.254,149.373
C00847=1111.597,47.785,-54.519,179.939,7.258,149.373
C00848=1111.592,48.034,-54.535,179.940,7.262,149.374
C00849=1111.587,48.285,-54.552,179.942,7.266,149.374
C00850=1111.582,48.534,-54.569,179.943,7.270,149.375
C00851=1111.577,48.783,-54.585,179.944,7.274,149.376
C00852=1111.573,49.032,-54.602,179.945,7.278,149.376
C00853=1111.568,49.281,-54.618,179.946,7.282,149.377
C00854=1111.562,49.531,-54.635,179.947,7.286,149.378
C00855=1111.558,49.745,-54.649,179.948,7.289,149.378
C00856=1111.554,49.959,-54.663,179.950,7.293,149.378
C00857=1111.550,50.173,-54.677,179.950,7.297,149.379
C00858=1111.545,50.387,-54.692,179.951,7.300,149.379
C00859=1111.541,50.602,-54.706,179.952,7.303,149.380
C00860=1111.537,50.816,-54.721,179.954,7.307,149.380
C00861=1111.533,51.030,-54.734,179.954,7.310,149.381
C00862=1111.528,51.244,-54.749,179.955,7.313,149.381
C00863=1111.524,51.494,-54.766,179.956,7.318,149.382
C00864=1111.519,51.743,-54.782,179.958,7.322,149.382
C00865=1111.514,51.992,-54.799,179.959,7.326,149.383
C00866=1111.509,52.242,-54.816,179.960,7.329,149.384
C00867=1111.504,52.491,-54.832,179.961,7.333,149.384
C00868=1111.499,52.740,-54.850,179.962,7.338,149.385
C00869=1111.494,52.990,-54.866,179.963,7.342,149.385
C00870=1111.489,53.239,-54.883,179.965,7.346,149.386
C00871=1111.484,53.489,-54.900,179.966,7.350,149.386
C00872=1111.479,53.738,-54.917,179.967,7.353,149.387
C00873=1111.475,53.988,-54.933,179.968,7.358,149.388
C00874=1111.469,54.237,-54.950,179.969,7.362,149.388
C00875=1111.465,54.486,-54.967,179.970,7.366,149.389
C00876=1111.459,54.736,-54.984,179.972,7.370,149.389
C00877=1111.454,54.985,-55.000,179.973,7.374,149.390
C00878=1111.450,55.234,-55.017,179.974,7.377,149.390
C00879=1111.445,55.484,-55.034,179.975,7.381,149.391
C00880=1111.440,55.733,-55.051,179.977,7.385,149.391
C00881=1111.434,55.983,-55.068,179.978,7.390,149.392
C00882=1111.430,56.231,-55.085,179.979,7.394,149.393
C00883=1111.425,56.481,-55.103,179.980,7.398,149.393
C00884=1111.421,56.731,-55.119,179.981,7.401,149.394
C00885=1111.415,56.980,-55.137,179.982,7.405,149.394
C00886=1111.410,57.229,-55.153,179.983,7.410,149.395
C00887=1111.405,57.479,-55.170,179.985,7.413,149.395
C00888=1111.401,57.728,-55.187,179.986,7.418,149.396
C00889=1111.396,57.978,-55.205,179.988,7.422,149.396
C00890=1111.391,58.226,-55.221,179.988,7.425,149.397
C00891=1111.385,58.476,-55.238,179.990,7.429,149.397
C00892=1111.381,58.726,-55.255,179.991,7.433,149.398
C00893=1111.376,58.975,-55.273,179.992,7.437,149.399
C00894=1111.371,59.224,-55.290,179.993,7.442,149.399
C00895=1111.366,59.474,-55.307,179.995,7.446,149.400
C00896=1111.361,59.723,-55.323,179.995,7.449,149.400
C00897=1111.356,59.972,-55.341,179.997,7.453,149.401
C00898=1111.352,60.222,-55.358,179.999,7.457,149.401
C00899=1111.347,60.471,-55.375,180.000,7.461,149.402
C00900=1111.342,60.721,-55.393,-179.999,7.465,149.402
C00901=1111.337,60.970,-55.410,-179.998,7.469,149.403
C00902=1111.331,61.219,-55.427,-179.997,7.472,149.403
C00903=1111.327,61.468,-55.444,-179.996,7.477,149.404
C00904=1111.322,61.718,-55.461,-179.994,7.481,149.404
C00905=1111.317,61.967,-55.478,-179.993,7.485,149.405
C00906=1111.313,62.217,-55.496,-179.991,7.489,149.405
C00907=1111.307,62.466,-55.513,-179.990,7.493,149.406
C00908=1111.303,62.715,-55.531,-179.989,7.497,149.407
C00909=1111.298,62.965,-55.548,-179.988,7.500,149.407
C00910=1111.292,63.214,-55.565,-179.987,7.504,149.408
C00911=1111.289,63.429,-55.580,-179.985,7.508,149.408
C00912=1111.284,63.643,-55.595,-179.984,7.511,149.409
C00913=1111.280,63.856,-55.609,-179.983,7.515,149.409
C00914=1111.276,64.070,-55.625,-179.982,7.519,149.409
C00915=1111.272,64.284,-55.639,-179.981,7.522,149.410
C00916=1111.267,64.498,-55.655,-179.980,7.525,149.410
C00917=1111.264,64.712,-55.669,-179.979,7.528,149.411
C00918=1111.259,64.926,-55.684,-179.977,7.532,149.411
C00919=1111.254,65.176,-55.702,-179.976,7.536,149.412
C00920=1111.250,65.425,-55.719,-179.975,7.540,149.412
C00921=1111.245,65.675,-55.736,-179.974,7.543,149.413
C00922=1111.240,65.924,-55.754,-179.973,7.547,149.413
C00923=1111.235,66.173,-55.772,-179.971,7.551,149.414
C00924=1111.230,66.423,-55.789,-179.970,7.556,149.414
C00925=1111.226,66.672,-55.807,-179.968,7.559,149.415
C00926=1111.220,66.922,-55.824,-179.967,7.563,149.415
C00927=1111.215,67.171,-55.842,-179.966,7.568,149.416
C00928=1111.211,67.420,-55.859,-179.965,7.571,149.416
C00929=1111.206,67.670,-55.877,-179.963,7.575,149.417
C00930=1111.201,67.919,-55.895,-179.962,7.579,149.417
C00931=1111.196,68.169,-55.912,-179.960,7.583,149.418
C00932=1111.191,68.417,-55.929,-179.959,7.587,149.418
C00933=1111.186,68.666,-55.947,-179.958,7.591,149.419
C00934=1111.181,68.916,-55.964,-179.956,7.595,149.419
C00935=1111.177,69.166,-55.983,-179.955,7.599,149.420
C00936=1111.172,69.415,-56.001,-179.953,7.603,149.420
C00937=1111.167,69.665,-56.018,-179.953,7.606,149.421
C00938=1111.162,69.913,-56.035,-179.951,7.611,149.422
C00939=1111.157,70.163,-56.053,-179.950,7.614,149.422
C00940=1111.152,70.412,-56.070,-179.948,7.618,149.422
C00941=1111.147,70.662,-56.088,-179.947,7.622,149.423
C00942=1111.142,70.911,-56.106,-179.946,7.627,149.423
C00943=1111.138,71.160,-56.124,-179.944,7.630,149.424
C00944=1111.132,71.410,-56.142,-179.942,7.634,149.424
C00945=1111.127,71.659,-56.160,-179.941,7.639,149.425
C00946=1111.123,71.908,-56.177,-179.940,7.642,149.425
C00947=1111.118,72.157,-56.195,-179.939,7.646,149.426
C00948=1111.113,72.406,-56.213,-179.938,7.650,149.426
C00949=1111.108,72.656,-56.230,-179.936,7.654,149.427
C00950=1111.103,72.905,-56.248,-179.935,7.658,149.427
C00951=1111.098,73.154,-56.266,-179.933,7.662,149.428
C00952=1111.093,73.403,-56.284,-179.932,7.666,149.428
C00953=1111.089,73.653,-56.303,-179.930,7.670,149.429
C00954=1111.084,73.902,-56.321,-179.929,7.674,149.429
C00955=1111.079,74.152,-56.339,-179.928,7.678,149.430
C00956=1111.074,74.401,-56.356,-179.926,7.682,149.430
C00957=1111.069,74.651,-56.374,-179.925,7.685,149.431
C00958=1111.064,74.900,-56.392,-179.924,7.689,149.431
C00959=1111.059,75.149,-56.410,-179.922,7.693,149.432
C00960=1111.054,75.398,-56.428,-179.921,7.697,149.432
C00961=1111.050,75.647,-56.446,-179.919,7.701,149.433
C00962=1111.045,75.897,-56.464,-179.918,7.705,149.433
C00963=1111.040,76.146,-56.482,-179.916,7.709,149.434
C00964=1111.035,76.396,-56.500,-179.915,7.713,149.434
C00965=1111.030,76.645,-56.518,-179.913,7.717,149.435
C00966=1111.026,76.894,-56.536,-179.912,7.721,149.435
C00967=1111.022,77.108,-56.552,-179.911,7.724,149.436
C00968=1111.017,77.322,-56.567,-179.910,7.728,149.436
C00969=1111.013,77.536,-56.583,-179.909,7.731,149.437
C00970=1111.008,77.750,-56.598,-179.909,7.734,149.437
C00971=1111.005,77.964,-56.614,-179.908,7.737,149.438
C00972=1111.001,78.177,-56.629,-179.907,7.740,149.438
C00973=1110.997,78.392,-56.645,-179.906,7.743,149.439
C00974=1110.992,78.605,-56.661,-179.905,7.747,149.439
C00975=1110.988,78.855,-56.679,-179.904,7.750,149.440
C00976=1110.983,79.104,-56.697,-179.903,7.754,149.440
C00977=1110.978,79.354,-56.715,-179.902,7.757,149.441
C00978=1110.973,79.603,-56.733,-179.901,7.762,149.441
C00979=1110.968,79.852,-56.751,-179.900,7.765,149.442
C00980=1110.963,80.101,-56.769,-179.899,7.769,149.443
C00981=1110.959,80.351,-56.788,-179.898,7.772,149.443
C00982=1110.954,80.600,-56.806,-179.897,7.777,149.444
C00983=1110.949,80.849,-56.824,-179.896,7.780,149.444
C00984=1110.944,81.098,-56.842,-179.895,7.784,149.445
C00985=1110.939,81.348,-56.861,-179.894,7.787,149.445
C00986=1110.934,81.598,-56.879,-179.893,7.791,149.446
C00987=1110.930,81.846,-56.898,-179.892,7.794,149.446
C00988=1110.925,82.095,-56.916,-179.891,7.799,149.447
C00989=1110.920,82.345,-56.934,-179.890,7.802,149.447
C00990=1110.915,82.595,-56.953,-179.889,7.806,149.448
C00991=1110.910,82.843,-56.972,-179.887,7.810,149.448
C00992=1110.905,83.092,-56.990,-179.887,7.814,149.449
C00993=1110.901,83.342,-57.008,-179.885,7.817,149.449
C00994=1110.896,83.591,-57.026,-179.885,7.821,149.450
C00995=1110.891,83.840,-57.045,-179.883,7.825,149.451
C00996=1110.886,84.090,-57.063,-179.882,7.829,149.451
C00997=1110.881,84.339,-57.081,-179.881,7.832,149.452
C00998=1110.876,84.589,-57.099,-179.880,7.836,149.452
C00999=1110.871,84.837,-57.119,-179.878,7.840,149.453
C01000=1110.867,85.087,-57.137,-179.877,7.843,149.453
C01001=1110.862,85.336,-57.155,-179.876,7.848,149.454
C01002=1110.857,85.585,-57.174,-179.875,7.851,149.454
C01003=1110.852,85.835,-57.193,-179.874,7.855,149.455
C01004=1110.847,86.084,-57.211,-179.872,7.859,149.455
C01005=1110.843,86.333,-57.229,-179.871,7.862,149.456
C01006=1110.837,86.582,-57.248,-179.870,7.866,149.456
C01007=1110.833,86.832,-57.267,-179.869,7.870,149.457
C01008=1110.828,87.081,-57.285,-179.868,7.874,149.457
C01009=1110.822,87.330,-57.304,-179.867,7.878,149.458
C01010=1110.818,87.580,-57.323,-179.865,7.882,149.458
C01011=1110.814,87.829,-57.341,-179.864,7.886,149.459
C01012=1110.809,88.078,-57.360,-179.863,7.889,149.459
C01013=1110.804,88.328,-57.378,-179.861,7.893,149.460
C01014=1110.799,88.576,-57.397,-179.860,7.897,149.460
C01015=1110.794,88.826,-57.416,-179.859,7.900,149.461
C01016=1110.790,89.075,-57.435,-179.858,7.904,149.461
C01017=1110.785,89.324,-57.453,-179.856,7.908,149.462
C01018=1110.780,89.574,-57.472,-179.855,7.912,149.462
C01019=1110.775,89.823,-57.490,-179.854,7.915,149.463
C01020=1110.770,90.072,-57.510,-179.852,7.919,149.463
C01021=1110.765,90.322,-57.528,-179.851,7.924,149.464
C01022=1110.761,90.570,-57.547,-179.850,7.927,149.464
C01023=1110.756,90.784,-57.563,-179.849,7.931,149.465
C01024=1110.752,90.999,-57.579,-179.848,7.934,149.465
C01025=1110.748,91.212,-57.595,-179.847,7.937,149.466
C01026=1110.744,91.426,-57.611,-179.846,7.940,149.466
C01027=1110.740,91.640,-57.627,-179.844,7.944,149.467
C01028=1110.736,91.854,-57.643,-179.843,7.947,149.467
C01029=1110.731,92.068,-57.660,-179.842,7.950,149.467
C01030=1110.728,92.282,-57.676,-179.841,7.953,149.468
C01031=1110.723,92.531,-57.694,-179.839,7.957,149.468
C01032=1110.718,92.780,-57.714,-179.838,7.961,149.469
C01033=1110.713,93.029,-57.732,-179.836,7.965,149.469
C01034=1110.708,93.278,-57.751,-179.835,7.969,149.470
C01035=1110.704,93.527,-57.770,-179.834,7.972,149.470
C01036=1110.698,93.777,-57.789,-179.832,7.976,149.470
C01037=1110.694,94.026,-57.808,-179.831,7.980,149.471
C01038=1110.689,94.275,-57.827,-179.829,7.983,149.471
C01039=1110.685,94.525,-57.846,-179.828,7.988,149.472
C01040=1110.679,94.774,-57.865,-179.826,7.992,149.472
C01041=1110.675,95.023,-57.885,-179.825,7.995,149.473
C01042=1110.670,95.272,-57.903,-179.824,7.999,149.473
C01043=1110.665,95.522,-57.922,-179.822,8.003,149.474
C01044=1110.660,95.771,-57.941,-179.820,8.006,149.474
C01045=1110.656,96.020,-57.961,-179.819,8.010,149.475
C01046=1110.651,96.269,-57.979,-179.817,8.014,149.475
C01047=1110.646,96.519,-57.998,-179.816,8.018,149.475
C01048=1110.641,96.768,-58.018,-179.815,8.021,149.476
C01049=1110.637,97.017,-58.037,-179.813,8.025,149.476
C01050=1110.631,97.266,-58.056,-179.812,8.029,149.477
C01051=1110.627,97.515,-58.075,-179.810,8.033,149.477
C01052=1110.622,97.764,-58.094,-179.808,8.037,149.478
C01053=1110.617,98.014,-58.114,-179.807,8.041,149.478
C01054=1110.612,98.263,-58.132,-179.805,8.044,149.478
C01055=1110.607,98.512,-58.152,-179.803,8.048,149.479
C01056=1110.603,98.762,-58.171,-179.803,8.051,149.479
C01057=1110.598,99.011,-58.190,-179.801,8.055,149.480
C01058=1110.593,99.260,-58.210,-179.799,8.059,149.480
C01059=1110.588,99.509,-58.229,-179.797,8.063,149.480
C01060=1110.584,99.758,-58.248,-179.796,8.067,149.481
C01061=1110.579,100.007,-58.267,-179.794,8.071,149.481
C01062=1110.574,100.257,-58.287,-179.792,8.074,149.482
C01063=1110.570,100.506,-58.306,-179.791,8.078,149.482
C01064=1110.565,100.755,-58.325,-179.789,8.082,149.483
C01065=1110.560,101.004,-58.345,-179.787,8.086,149.483
C01066=1110.554,101.253,-58.364,-179.786,8.090,149.483
C01067=1110.550,101.502,-58.383,-179.784,8.093,149.484
C01068=1110.546,101.752,-58.403,-179.782,8.097,149.484
C01069=1110.540,102.001,-58.422,-179.780,8.101,149.484
C01070=1110.536,102.251,-58.442,-179.779,8.104,149.485
C01071=1110.532,102.500,-58.461,-179.778,8.108,149.485
C01072=1110.526,102.749,-58.480,-179.776,8.112,149.486
C01073=1110.522,102.998,-58.500,-179.774,8.115,149.486
C01074=1110.516,103.247,-58.519,-179.772,8.119,149.486
C01075=1110.511,103.497,-58.539,-179.771,8.123,149.487
C01076=1110.508,103.745,-58.559,-179.769,8.127,149.487
C01077=1110.502,103.994,-58.578,-179.767,8.130,149.487
C01078=1110.498,104.244,-58.598,-179.766,8.134,149.488
C01079=1110.493,104.458,-58.614,-179.764,8.138,149.488
C01080=1110.490,104.672,-58.631,-179.762,8.141,149.488
C01081=1110.485,104.885,-58.648,-179.761,8.144,149.489
C01082=1110.482,105.099,-58.665,-179.759,8.147,149.489
C01083=1110.477,105.313,-58.682,-179.758,8.150,149.489
C01084=1110.473,105.526,-58.698,-179.756,8.154,149.490
C01085=1110.469,105.740,-58.715,-179.755,8.156,149.490
C01086=1110.465,105.954,-58.732,-179.753,8.160,149.490
C01087=1110.460,106.203,-58.752,-179.751,8.164,149.490
C01088=1110.455,106.452,-58.771,-179.749,8.167,149.491
C01089=1110.451,106.701,-58.791,-179.747,8.171,149.491
C01090=1110.446,106.951,-58.811,-179.745,8.175,149.491
C01091=1110.441,107.200,-58.831,-179.744,8.179,149.492
C01092=1110.436,107.449,-58.851,-179.742,8.182,149.492
C01093=1110.431,107.698,-58.870,-179.740,8.186,149.492
C01094=1110.427,107.948,-58.890,-179.738,8.190,149.493
C01095=1110.422,108.197,-58.910,-179.736,8.193,149.493
C01096=1110.417,108.446,-58.930,-179.734,8.197,149.493
C01097=1110.412,108.695,-58.949,-179.732,8.200,149.494
C01098=1110.408,108.944,-58.970,-179.730,8.204,149.494
C01099=1110.403,109.194,-58.989,-179.729,8.208,149.494
C01100=1110.398,109.443,-59.009,-179.726,8.211,149.494
C01101=1110.393,109.692,-59.029,-179.724,8.215,149.495
C01102=1110.388,109.941,-59.049,-179.723,8.219,149.495
C01103=1110.384,110.190,-59.069,-179.721,8.222,149.495
C01104=1110.379,110.440,-59.089,-179.719,8.226,149.496
C01105=1110.374,110.688,-59.109,-179.717,8.229,149.496
C01106=1110.369,110.937,-59.128,-179.715,8.233,149.496
C01107=1110.365,111.186,-59.149,-179.713,8.237,149.496
C01108=1110.360,111.436,-59.168,-179.711,8.240,149.497
C01109=1110.356,111.685,-59.189,-179.709,8.244,149.497
C01110=1110.350,111.934,-59.208,-179.708,8.247,149.497
C01111=1110.346,112.183,-59.228,-179.706,8.250,149.498
C01112=1110.341,112.432,-59.248,-179.704,8.254,149.498
C01113=1110.337,112.681,-59.268,-179.702,8.258,149.498
C01114=1110.332,112.931,-59.288,-179.701,8.260,149.498
C01115=1110.327,113.180,-59.309,-179.699,8.264,149.499
C01116=1110.322,113.430,-59.329,-179.697,8.268,149.499
C01117=1110.317,113.678,-59.349,-179.695,8.271,149.499
C01118=1110.313,113.927,-59.369,-179.694,8.274,149.500
C01119=1110.308,114.176,-59.389,-179.692,8.278,149.500
C01120=1110.303,114.425,-59.409,-179.690,8.281,149.500
C01121=1110.299,114.675,-59.429,-179.689,8.284,149.501
C01122=1110.294,114.924,-59.450,-179.687,8.288,149.501
C01123=1110.289,115.173,-59.470,-179.685,8.291,149.501
C01124=1110.284,115.423,-59.490,-179.683,8.295,149.502
C01125=1110.279,115.671,-59.510,-179.682,8.298,149.502
C01126=1110.275,115.920,-59.530,-179.680,8.301,149.502
C01127=1110.269,116.170,-59.550,-179.678,8.305,149.502
C01128=1110.265,116.419,-59.571,-179.676,8.309,149.503
C01129=1110.261,116.668,-59.591,-179.675,8.312,149.503
C01130=1110.256,116.917,-59.611,-179.672,8.315,149.503
C01131=1110.251,117.166,-59.632,-179.671,8.319,149.504
C01132=1110.246,117.415,-59.652,-179.669,8.322,149.504
C01133=1110.242,117.664,-59.672,-179.667,8.325,149.504
C01134=1110.237,117.913,-59.693,-179.666,8.329,149.504
C01135=1110.233,118.127,-59.710,-179.664,8.332,149.505
C01136=1110.229,118.341,-59.728,-179.663,8.334,149.505
C01137=1110.225,118.555,-59.745,-179.661,8.337,149.505
C01138=1110.220,118.768,-59.762,-179.659,8.341,149.505
C01139=1110.216,118.982,-59.781,-179.658,8.343,149.506
C01140=1110.213,119.195,-59.797,-179.656,8.346,149.506
C01141=1110.209,119.409,-59.815,-179.655,8.349,149.506
C01142=1110.204,119.623,-59.832,-179.654,8.352,149.506
C01143=1110.199,119.872,-59.853,-179.652,8.355,149.507
C01144=1110.195,120.121,-59.874,-179.650,8.359,149.507
C01145=1110.190,120.370,-59.894,-179.648,8.362,149.507
C01146=1110.186,120.619,-59.914,-179.646,8.365,149.507
C01147=1110.181,120.868,-59.935,-179.645,8.369,149.508
C01148=1110.176,121.117,-59.956,-179.643,8.372,149.508
C01149=1110.171,121.366,-59.977,-179.641,8.375,149.508
C01150=1110.167,121.615,-59.997,-179.639,8.379,149.509
C01151=1110.162,121.864,-60.017,-179.638,8.383,149.509
C01152=1110.157,122.113,-60.038,-179.636,8.385,149.509
C01153=1110.153,122.362,-60.059,-179.634,8.389,149.509
C01154=1110.148,122.612,-60.078,-179.632,8.392,149.510
C01155=1110.143,122.861,-60.100,-179.631,8.395,149.510
C01156=1110.139,123.110,-60.121,-179.629,8.399,149.510
C01157=1110.134,123.359,-60.142,-179.627,8.402,149.511
C01158=1110.130,123.608,-60.162,-179.625,8.405,149.511
C01159=1110.125,123.857,-60.182,-179.624,8.409,149.511
C01160=1110.120,124.107,-60.203,-179.622,8.412,149.511
C01161=1110.116,124.356,-60.224,-179.620,8.415,149.512
C01162=1110.110,124.605,-60.245,-179.618,8.419,149.512
C01163=1110.106,124.854,-60.265,-179.617,8.423,149.512
C01164=1110.101,125.103,-60.286,-179.615,8.425,149.513
C01165=1110.096,125.352,-60.306,-179.613,8.429,149.513
C01166=1110.091,125.601,-60.327,-179.611,8.432,149.513
C01167=1110.087,125.850,-60.348,-179.610,8.435,149.513
C01168=1110.082,126.100,-60.370,-179.608,8.439,149.514
C01169=1110.078,126.349,-60.390,-179.606,8.442,149.514
C01170=1110.073,126.598,-60.411,-179.604,8.446,149.514
C01171=1110.068,126.847,-60.432,-179.602,8.449,149.514
C01172=1110.063,127.096,-60.453,-179.601,8.452,149.515
C01173=1110.059,127.345,-60.473,-179.599,8.456,149.515
C01174=1110.054,127.594,-60.495,-179.597,8.459,149.515
C01175=1110.049,127.843,-60.515,-179.595,8.462,149.515
C01176=1110.045,128.092,-60.536,-179.594,8.466,149.516
C01177=1110.040,128.342,-60.557,-179.592,8.469,149.516
C01178=1110.036,128.590,-60.578,-179.590,8.472,149.516
C01179=1110.030,128.839,-60.599,-179.588,8.476,149.517
C01180=1110.026,129.088,-60.620,-179.587,8.479,149.517
C01181=1110.021,129.338,-60.641,-179.585,8.482,149.517
C01182=1110.016,129.586,-60.662,-179.583,8.486,149.518
C01183=1110.012,129.836,-60.683,-179.581,8.489,149.518
C01184=1110.007,130.085,-60.704,-179.580,8.492,149.518
C01185=1110.003,130.333,-60.725,-179.578,8.496,149.518
C01186=1109.998,130.583,-60.746,-179.576,8.499,149.519
C01187=1109.992,130.832,-60.767,-179.574,8.502,149.519
C01188=1109.989,131.081,-60.789,-179.573,8.506,149.519
C01189=1109.984,131.330,-60.809,-179.571,8.509,149.520
C01190=1109.979,131.579,-60.830,-179.569,8.512,149.520
C01191=1109.975,131.793,-60.849,-179.568,8.515,149.520
C01192=1109.971,132.006,-60.867,-179.566,8.518,149.520
C01193=1109.967,132.220,-60.885,-179.565,8.522,149.521
C01194=1109.963,132.433,-60.903,-179.563,8.524,149.521
C01195=1109.958,132.647,-60.921,-179.562,8.527,149.521
C01196=1109.954,132.860,-60.939,-179.560,8.530,149.521
C01197=1109.951,133.074,-60.958,-179.559,8.532,149.522
C01198=1109.947,133.288,-60.975,-179.557,8.535,149.522
C01199=1109.942,133.536,-60.997,-179.555,8.539,149.522
C01200=1109.937,133.786,-61.018,-179.554,8.542,149.522
C01201=1109.933,134.035,-61.040,-179.552,8.545,149.523
C01202=1109.928,134.284,-61.060,-179.550,8.549,149.523
C01203=1109.923,134.533,-61.082,-179.548,8.552,149.523
C01204=1109.919,134.783,-61.103,-179.547,8.555,149.524
C01205=1109.914,135.031,-61.125,-179.545,8.559,149.524
C01206=1109.910,135.280,-61.146,-179.543,8.562,149.524
C01207=1109.904,135.529,-61.167,-179.542,8.565,149.525
C01208=1109.900,135.778,-61.189,-179.540,8.569,149.525
C01209=1109.895,136.027,-61.210,-179.538,8.572,149.525
C01210=1109.891,136.276,-61.231,-179.536,8.576,149.525
C01211=1109.886,136.526,-61.253,-179.535,8.579,149.526
C01212=1109.881,136.774,-61.274,-179.533,8.582,149.526
C01213=1109.877,137.023,-61.296,-179.531,8.586,149.526
C01214=1109.871,137.272,-61.317,-179.530,8.589,149.527
C01215=1109.867,137.522,-61.339,-179.528,8.592,149.527
C01216=1109.863,137.770,-61.360,-179.526,8.596,149.527
C01217=1109.858,138.019,-61.381,-179.524,8.599,149.527
C01218=1109.854,138.268,-61.403,-179.522,8.603,149.528
C01219=1109.849,138.517,-61.425,-179.521,8.606,149.528
C01220=1109.844,138.767,-61.446,-179.519,8.609,149.528
C01221=1109.839,139.016,-61.468,-179.517,8.613,149.529
C01222=1109.834,139.264,-61.489,-179.516,8.616,149.529
C01223=1109.830,139.514,-61.512,-179.513,8.620,149.529
C01224=1109.826,139.763,-61.532,-179.512,8.623,149.529
C01225=1109.821,140.011,-61.554,-179.510,8.627,149.530
C01226=1109.817,140.261,-61.576,-179.508,8.630,149.530
C01227=1109.812,140.509,-61.597,-179.507,8.633,149.531
C01228=1109.806,140.759,-61.618,-179.505,8.637,149.531
C01229=1109.802,141.008,-61.640,-179.503,8.640,149.531
C01230=1109.797,141.257,-61.662,-179.502,8.643,149.532
C01231=1109.793,141.506,-61.684,-179.500,8.647,149.532
C01232=1109.788,141.754,-61.706,-179.498,8.651,149.532
C01233=1109.784,142.004,-61.728,-179.496,8.654,149.532
C01234=1109.779,142.253,-61.749,-179.495,8.657,149.533
C01235=1109.774,142.502,-61.770,-179.493,8.661,149.533
C01236=1109.770,142.751,-61.792,-179.491,8.664,149.533
C01237=1109.765,143.000,-61.814,-179.490,8.667,149.534
C01238=1109.760,143.249,-61.836,-179.488,8.671,149.534
C01239=1109.756,143.498,-61.858,-179.486,8.675,149.534
C01240=1109.751,143.747,-61.880,-179.484,8.678,149.535
C01241=1109.746,143.996,-61.902,-179.483,8.681,149.535
C01242=1109.742,144.244,-61.923,-179.481,8.685,149.535
C01243=1109.737,144.494,-61.945,-179.480,8.689,149.536
C01244=1109.732,144.742,-61.967,-179.478,8.691,149.536
C01245=1109.728,144.992,-61.989,-179.476,8.695,149.536
C01246=1109.723,145.240,-62.011,-179.475,8.699,149.537
C01247=1109.719,145.454,-62.030,-179.473,8.701,149.537
C01248=1109.715,145.668,-62.048,-179.471,8.705,149.537
C01249=1109.711,145.882,-62.067,-179.470,8.707,149.537
C01250=1109.708,146.094,-62.086,-179.467,8.711,149.538
C01251=1109.703,146.308,-62.105,-179.466,8.714,149.538
C01252=1109.700,146.522,-62.123,-179.464,8.717,149.538
C01253=1109.695,146.735,-62.143,-179.463,8.720,149.539
C01254=1109.692,146.948,-62.161,-179.461,8.723,149.539
C01255=1109.686,147.197,-62.183,-179.459,8.726,149.539
C01256=1109.682,147.447,-62.205,-179.457,8.730,149.539
C01257=1109.677,147.695,-62.227,-179.455,8.733,149.539
C01258=1109.673,147.945,-62.249,-179.453,8.737,149.540
C01259=1109.668,148.193,-62.271,-179.451,8.740,149.540
C01260=1109.664,148.442,-62.294,-179.449,8.744,149.540
C01261=1109.659,148.692,-62.316,-179.447,8.748,149.541
C01262=1109.654,148.940,-62.338,-179.445,8.751,149.541
C01263=1109.650,149.190,-62.360,-179.443,8.755,149.541
C01264=1109.645,149.438,-62.382,-179.441,8.758,149.541
C01265=1109.641,149.688,-62.404,-179.439,8.762,149.542
C01266=1109.635,149.936,-62.427,-179.437,8.765,149.542
C01267=1109.631,150.185,-62.449,-179.435,8.769,149.542
C01268=1109.626,150.434,-62.470,-179.433,8.772,149.542
C01269=1109.622,150.683,-62.492,-179.431,8.776,149.543
C01270=1109.617,150.932,-62.516,-179.429,8.779,149.543
C01271=1109.612,151.181,-62.537,-179.427,8.783,149.543
C01272=1109.608,151.430,-62.560,-179.424,8.786,149.543
C01273=1109.604,151.678,-62.582,-179.423,8.789,149.543
C01274=1109.599,151.928,-62.605,-179.421,8.792,149.544
C01275=1109.594,152.177,-62.627,-179.419,8.796,149.544
C01276=1109.589,152.426,-62.648,-179.416,8.799,149.544
C01277=1109.585,152.675,-62.672,-179.414,8.802,149.544
C01278=1109.580,152.924,-62.693,-179.412,8.806,149.544
C01279=1109.576,153.172,-62.716,-179.410,8.809,149.545
C01280=1109.571,153.422,-62.739,-179.408,8.813,149.545
C01281=1109.566,153.671,-62.760,-179.406,8.816,149.545
C01282=1109.562,153.919,-62.783,-179.404,8.819,149.545
C01283=1109.557,154.169,-62.806,-179.402,8.822,149.545
C01284=1109.553,154.417,-62.828,-179.400,8.826,149.546
C01285=1109.548,154.667,-62.851,-179.398,8.829,149.546
C01286=1109.544,154.915,-62.874,-179.396,8.833,149.546
C01287=1109.539,155.164,-62.895,-179.394,8.836,149.546
C01288=1109.534,155.414,-62.918,-179.391,8.839,149.546
C01289=1109.530,155.662,-62.941,-179.390,8.842,149.547
C01290=1109.524,155.911,-62.963,-179.388,8.845,149.547
C01291=1109.520,156.160,-62.986,-179.386,8.849,149.547
C01292=1109.516,156.409,-63.008,-179.383,8.852,149.547
C01293=1109.511,156.658,-63.031,-179.381,8.856,149.547
C01294=1109.507,156.906,-63.054,-179.379,8.858,149.548
C01295=1109.502,157.156,-63.076,-179.377,8.861,149.548
C01296=1109.498,157.405,-63.099,-179.375,8.865,149.548
C01297=1109.492,157.654,-63.121,-179.373,8.868,149.548
C01298=1109.488,157.903,-63.144,-179.370,8.871,149.548
C01299=1109.483,158.152,-63.167,-179.368,8.875,149.548
C01300=1109.479,158.400,-63.189,-179.367,8.878,149.549
C01301=1109.474,158.649,-63.212,-179.364,8.881,149.549
C01302=1109.470,158.899,-63.234,-179.362,8.884,149.549
C01303=1109.466,159.112,-63.254,-179.361,8.887,149.549
C01304=1109.461,159.325,-63.274,-179.359,8.889,149.549
C01305=1109.458,159.539,-63.294,-179.357,8.893,149.549
C01306=1109.454,159.752,-63.313,-179.355,8.895,149.549
C01307=1109.450,159.965,-63.332,-179.353,8.898,149.550
C01308=1109.446,160.178,-63.352,-179.351,8.900,149.550
C01309=1109.443,160.392,-63.372,-179.349,8.904,149.550
C01310=1109.438,160.605,-63.391,-179.347,8.906,149.550
C01311=1109.433,160.854,-63.414,-179.345,8.909,149.550
C01312=1109.429,161.103,-63.437,-179.343,8.912,149.550
C01313=1109.425,161.352,-63.460,-179.341,8.915,149.550
C01314=1109.420,161.600,-63.482,-179.339,8.918,149.551
C01315=1109.415,161.850,-63.505,-179.337,8.922,149.551
C01316=1109.410,162.099,-63.528,-179.335,8.924,149.551
C01317=1109.406,162.347,-63.551,-179.333,8.928,149.551
C01318=1109.402,162.596,-63.574,-179.330,8.931,149.551
C01319=1109.397,162.846,-63.598,-179.328,8.934,149.551
C01320=1109.392,163.094,-63.620,-179.326,8.937,149.551
C01321=1109.387,163.343,-63.643,-179.324,8.940,149.552
C01322=1109.383,163.592,-63.666,-179.322,8.943,149.552
C01323=1109.379,163.841,-63.689,-179.320,8.946,149.552
C01324=1109.374,164.090,-63.712,-179.318,8.949,149.552
C01325=1109.370,164.339,-63.735,-179.316,8.952,149.552
C01326=1109.365,164.588,-63.758,-179.313,8.956,149.552
C01327=1109.360,164.836,-63.781,-179.312,8.958,149.552
C01328=1109.356,165.085,-63.804,-179.309,8.961,149.552
C01329=1109.351,165.334,-63.828,-179.307,8.965,149.553
C01330=1109.347,165.583,-63.851,-179.305,8.967,149.553
C01331=1109.342,165.832,-63.874,-179.303,8.970,149.553
C01332=1109.338,166.081,-63.897,-179.301,8.974,149.553
C01333=1109.333,166.330,-63.920,-179.298,8.977,149.553
C01334=1109.329,166.579,-63.944,-179.297,8.980,149.553
C01335=1109.324,166.828,-63.967,-179.294,8.983,149.553
C01336=1109.319,167.076,-63.990,-179.292,8.986,149.553
C01337=1109.315,167.325,-64.013,-179.290,8.989,149.554
C01338=1109.310,167.574,-64.036,-179.288,8.992,149.554
C01339=1109.305,167.823,-64.060,-179.285,8.995,149.554
C01340=1109.301,168.072,-64.083,-179.284,8.998,149.554
C01341=1109.297,168.321,-64.106,-179.281,9.001,149.554
C01342=1109.292,168.570,-64.129,-179.279,9.004,149.554
C01343=1109.287,168.819,-64.152,-179.276,9.007,149.554
C01344=1109.283,169.068,-64.176,-179.275,9.010,149.554
C01345=1109.278,169.317,-64.199,-179.273,9.013,149.554
C01346=1109.273,169.565,-64.223,-179.270,9.016,149.555
C01347=1109.269,169.814,-64.247,-179.269,9.019,149.555
C01348=1109.265,170.063,-64.269,-179.266,9.022,149.555
C01349=1109.260,170.312,-64.293,-179.263,9.025,149.555
C01350=1109.255,170.561,-64.316,-179.262,9.028,149.555
C01351=1109.251,170.809,-64.340,-179.260,9.031,149.555
C01352=1109.246,171.058,-64.364,-179.257,9.034,149.555
C01353=1109.242,171.307,-64.387,-179.256,9.037,149.555
C01354=1109.237,171.556,-64.410,-179.253,9.040,149.555
C01355=1109.232,171.805,-64.434,-179.250,9.043,149.555
C01356=1109.228,172.054,-64.458,-179.249,9.046,149.556
C01357=1109.223,172.303,-64.481,-179.246,9.049,149.556
C01358=1109.219,172.552,-64.504,-179.244,9.052,149.556
C01359=1109.215,172.765,-64.525,-179.243,9.055,149.556
C01360=1109.211,172.978,-64.544,-179.241,9.057,149.556
C01361=1109.207,173.191,-64.565,-179.239,9.059,149.556
C01362=1109.203,173.404,-64.585,-179.237,9.062,149.556
C01363=1109.199,173.617,-64.606,-179.235,9.064,149.556
C01364=1109.195,173.831,-64.626,-179.233,9.067,149.556
C01365=1109.192,174.045,-64.645,-179.231,9.070,149.556
C01366=1109.188,174.258,-64.666,-179.230,9.072,149.557
C01367=1109.183,174.507,-64.689,-179.228,9.075,149.557
C01368=1109.179,174.755,-64.713,-179.225,9.078,149.557
C01369=1109.174,175.004,-64.737,-179.223,9.081,149.557
C01370=1109.170,175.252,-64.761,-179.221,9.084,149.557
C01371=1109.165,175.501,-64.784,-179.219,9.087,149.557
C01372=1109.161,175.750,-64.807,-179.217,9.090,149.557
C01373=1109.155,175.999,-64.832,-179.215,9.093,149.557
C01374=1109.151,176.248,-64.856,-179.212,9.096,149.557
C01375=1109.146,176.497,-64.880,-179.210,9.099,149.557
C01376=1109.142,176.746,-64.903,-179.208,9.102,149.558
C01377=1109.138,176.995,-64.927,-179.206,9.105,149.558
C01378=1109.133,177.244,-64.951,-179.203,9.108,149.558
C01379=1109.129,177.492,-64.975,-179.202,9.110,149.558
C01380=1109.124,177.741,-64.998,-179.199,9.114,149.558
C01381=1109.120,177.990,-65.022,-179.197,9.117,149.558
C01382=1109.115,178.238,-65.046,-179.195,9.119,149.558
C01383=1109.111,178.487,-65.070,-179.193,9.122,149.558
C01384=1109.107,178.736,-65.094,-179.190,9.126,149.558
C01385=1109.101,178.986,-65.118,-179.189,9.128,149.559
C01386=1109.097,179.234,-65.142,-179.186,9.131,149.559
C01387=1109.092,179.482,-65.166,-179.184,9.135,149.559
C01388=1109.088,179.731,-65.190,-179.182,9.137,149.559
C01389=1109.083,179.980,-65.214,-179.180,9.140,149.559
C01390=1109.079,180.230,-65.237,-179.177,9.143,149.559
C01391=1109.074,180.478,-65.262,-179.175,9.147,149.559
C01392=1109.070,180.727,-65.286,-179.172,9.150,149.559
C01393=1109.065,180.976,-65.309,-179.170,9.152,149.559
C01394=1109.061,181.224,-65.334,-179.168,9.155,149.559
C01395=1109.057,181.473,-65.358,-179.165,9.159,149.559
C01396=1109.052,181.722,-65.382,-179.163,9.162,149.560
C01397=1109.047,181.971,-65.406,-179.161,9.164,149.560
C01398=1109.043,182.219,-65.430,-179.159,9.167,149.560
C01399=1109.038,182.468,-65.454,-179.156,9.170,149.560
C01400=1109.034,182.717,-65.479,-179.154,9.173,149.560
C01401=1109.029,182.966,-65.503,-179.152,9.176,149.560
C01402=1109.025,183.215,-65.527,-179.149,9.179,149.560
C01403=1109.020,183.463,-65.551,-179.147,9.182,149.560
C01404=1109.016,183.713,-65.576,-179.144,9.185,149.560
C01405=1109.011,183.961,-65.600,-179.142,9.187,149.560
C01406=1109.007,184.209,-65.624,-179.140,9.190,149.560
C01407=1109.001,184.459,-65.648,-179.137,9.194,149.560
C01408=1108.998,184.708,-65.672,-179.135,9.196,149.560
C01409=1108.993,184.956,-65.696,-179.133,9.199,149.560
C01410=1108.989,185.205,-65.720,-179.130,9.202,149.560
C01411=1108.984,185.453,-65.745,-179.128,9.204,149.560
C01412=1108.980,185.703,-65.770,-179.126,9.208,149.560
C01413=1108.975,185.951,-65.794,-179.123,9.211,149.560
C01414=1108.970,186.200,-65.818,-179.121,9.213,149.560
C01415=1108.967,186.413,-65.839,-179.119,9.216,149.560
C01416=1108.963,186.626,-65.860,-179.117,9.218,149.560
C01417=1108.959,186.840,-65.881,-179.115,9.221,149.560
C01418=1108.956,187.053,-65.902,-179.113,9.223,149.560
C01419=1108.952,187.266,-65.923,-179.111,9.225,149.561
C01420=1108.947,187.479,-65.944,-179.109,9.228,149.561
C01421=1108.944,187.692,-65.965,-179.107,9.230,149.561
C01422=1108.940,187.905,-65.986,-179.106,9.232,149.561
C01423=1108.935,188.154,-66.010,-179.103,9.236,149.561
C01424=1108.930,188.403,-66.035,-179.101,9.239,149.561
C01425=1108.926,188.652,-66.059,-179.099,9.241,149.561
C01426=1108.921,188.900,-66.084,-179.096,9.244,149.561
C01427=1108.917,189.149,-66.108,-179.094,9.246,149.561
C01428=1108.913,189.398,-66.133,-179.092,9.250,149.561
C01429=1108.908,189.646,-66.158,-179.089,9.253,149.561
C01430=1108.904,189.895,-66.183,-179.087,9.255,149.561
C01431=1108.899,190.144,-66.207,-179.085,9.258,149.561
C01432=1108.894,190.393,-66.231,-179.083,9.260,149.561
C01433=1108.890,190.642,-66.256,-179.080,9.264,149.561
C01434=1108.885,190.890,-66.280,-179.078,9.267,149.561
C01435=1108.881,191.138,-66.305,-179.076,9.269,149.561
C01436=1108.877,191.388,-66.330,-179.073,9.272,149.561
C01437=1108.872,191.636,-66.354,-179.072,9.274,149.561
C01438=1108.868,191.885,-66.379,-179.069,9.278,149.561
C01439=1108.863,192.134,-66.403,-179.066,9.281,149.561
C01440=1108.859,192.383,-66.429,-179.065,9.283,149.561
C01441=1108.855,192.631,-66.453,-179.062,9.286,149.561
C01442=1108.849,192.880,-66.478,-179.060,9.288,149.562
C01443=1108.845,193.129,-66.503,-179.058,9.292,149.562
C01444=1108.841,193.377,-66.528,-179.056,9.294,149.562
C01445=1108.836,193.626,-66.553,-179.054,9.297,149.562
C01446=1108.832,193.875,-66.577,-179.051,9.300,149.562
C01447=1108.828,194.124,-66.603,-179.049,9.303,149.562
C01448=1108.823,194.372,-66.627,-179.047,9.306,149.562
C01449=1108.818,194.621,-66.651,-179.045,9.308,149.562
C01450=1108.814,194.870,-66.677,-179.042,9.311,149.562
C01451=1108.809,195.118,-66.702,-179.040,9.315,149.562
C01452=1108.805,195.367,-66.726,-179.038,9.317,149.562
C01453=1108.800,195.616,-66.752,-179.036,9.320,149.562
C01454=1108.796,195.865,-66.777,-179.034,9.323,149.562
C01455=1108.792,196.113,-66.801,-179.032,9.326,149.563
C01456=1108.787,196.362,-66.826,-179.029,9.329,149.563
C01457=1108.782,196.611,-66.851,-179.027,9.332,149.563
C01458=1108.778,196.859,-66.876,-179.025,9.335,149.563
C01459=1108.773,197.108,-66.901,-179.022,9.338,149.563
C01460=1108.769,197.357,-66.927,-179.020,9.341,149.563
C01461=1108.765,197.605,-66.951,-179.017,9.344,149.563
C01462=1108.760,197.854,-66.977,-179.015,9.347,149.563
C01463=1108.755,198.103,-67.001,-179.013,9.349,149.563
C01464=1108.751,198.352,-67.027,-179.010,9.352,149.563
C01465=1108.747,198.601,-67.051,-179.008,9.356,149.563
C01466=1108.742,198.849,-67.077,-179.005,9.358,149.563
C01467=1108.738,199.098,-67.102,-179.002,9.361,149.563
C01468=1108.733,199.346,-67.127,-179.000,9.365,149.563
C01469=1108.730,199.595,-67.152,-178.997,9.367,149.563
C01470=1108.725,199.844,-67.177,-178.994,9.370,149.563
C01471=1108.721,200.057,-67.199,-178.992,9.373,149.563
C01472=1108.717,200.270,-67.220,-178.990,9.375,149.563
C01473=1108.713,200.483,-67.242,-178.988,9.378,149.563
C01474=1108.709,200.695,-67.264,-178.986,9.380,149.563
C01475=1108.706,200.909,-67.285,-178.983,9.382,149.563
C01476=1108.702,201.122,-67.307,-178.981,9.385,149.563
C01477=1108.698,201.335,-67.329,-178.979,9.387,149.563
C01478=1108.694,201.549,-67.351,-178.977,9.390,149.563
C01479=1108.689,201.797,-67.376,-178.974,9.392,149.563
C01480=1108.685,202.046,-67.402,-178.971,9.395,149.563
C01481=1108.681,202.295,-67.426,-178.968,9.398,149.563
C01482=1108.677,202.543,-67.452,-178.966,9.401,149.563
C01483=1108.672,202.792,-67.477,-178.963,9.404,149.563
C01484=1108.667,203.040,-67.503,-178.960,9.407,149.562
C01485=1108.663,203.289,-67.528,-178.957,9.410,149.562
C01486=1108.659,203.538,-67.553,-178.954,9.413,149.562
C01487=1108.654,203.786,-67.579,-178.951,9.415,149.562
C01488=1108.650,204.035,-67.605,-178.949,9.418,149.562
C01489=1108.645,204.284,-67.630,-178.946,9.421,149.562
C01490=1108.641,204.532,-67.656,-178.943,9.424,149.562
C01491=1108.636,204.781,-67.681,-178.940,9.427,149.562
C01492=1108.632,205.030,-67.707,-178.938,9.430,149.562
C01493=1108.627,205.278,-67.732,-178.935,9.433,149.562
C01494=1108.623,205.527,-67.758,-178.932,9.435,149.562
C01495=1108.619,205.776,-67.783,-178.929,9.438,149.562
C01496=1108.614,206.024,-67.809,-178.925,9.442,149.562
C01497=1108.610,206.273,-67.835,-178.923,9.445,149.561
C01498=1108.605,206.521,-67.860,-178.920,9.447,149.561
C01499=1108.601,206.770,-67.886,-178.917,9.450,149.561
C01500=1108.596,207.018,-67.911,-178.914,9.453,149.561
C01501=1108.592,207.267,-67.937,-178.911,9.456,149.561
C01502=1108.588,207.516,-67.963,-178.908,9.459,149.561
C01503=1108.583,207.764,-67.988,-178.905,9.461,149.561
C01504=1108.579,208.013,-68.014,-178.902,9.465,149.561
C01505=1108.574,208.262,-68.040,-178.899,9.468,149.561
C01506=1108.570,208.511,-68.066,-178.896,9.471,149.561
C01507=1108.565,208.760,-68.092,-178.893,9.474,149.560
C01508=1108.561,209.008,-68.117,-178.890,9.477,149.560
C01509=1108.556,209.256,-68.143,-178.887,9.480,149.560
C01510=1108.552,209.505,-68.169,-178.884,9.483,149.560
C01511=1108.548,209.753,-68.195,-178.881,9.486,149.560
C01512=1108.543,210.002,-68.221,-178.878,9.490,149.560
C01513=1108.538,210.251,-68.247,-178.875,9.492,149.560
C01514=1108.534,210.499,-68.273,-178.872,9.495,149.560
C01515=1108.530,210.748,-68.299,-178.869,9.499,149.560
C01516=1108.526,210.996,-68.325,-178.866,9.502,149.560
C01517=1108.521,211.246,-68.351,-178.863,9.505,149.560
C01518=1108.516,211.494,-68.377,-178.860,9.508,149.560
C01519=1108.512,211.742,-68.402,-178.856,9.512,149.560
C01520=1108.508,211.991,-68.429,-178.854,9.515,149.560
C01521=1108.504,212.239,-68.455,-178.851,9.518,149.560
C01522=1108.499,212.489,-68.481,-178.847,9.521,149.559
C01523=1108.495,212.737,-68.508,-178.845,9.524,149.559
C01524=1108.491,212.986,-68.533,-178.841,9.528,149.559
C01525=1108.485,213.234,-68.559,-178.838,9.532,149.559
C01526=1108.481,213.482,-68.586,-178.835,9.535,149.559
C01527=1108.478,213.695,-68.608,-178.834,9.537,149.560
C01528=1108.473,213.908,-68.630,-178.831,9.540,149.560
C01529=1108.470,214.122,-68.653,-178.829,9.543,149.560
C01530=1108.466,214.334,-68.675,-178.827,9.545,149.560
C01531=1108.462,214.547,-68.698,-178.826,9.547,149.560
C01532=1108.458,214.760,-68.720,-178.824,9.550,149.560
C01533=1108.455,214.973,-68.743,-178.822,9.552,149.560
C01534=1108.451,215.186,-68.765,-178.820,9.555,149.560
C01535=1108.447,215.434,-68.791,-178.818,9.558,149.560
C01536=1108.443,215.683,-68.817,-178.815,9.561,149.560
C01537=1108.438,215.932,-68.844,-178.813,9.564,149.560
C01538=1108.434,216.180,-68.870,-178.811,9.568,149.561
C01539=1108.429,216.428,-68.897,-178.809,9.570,149.561
C01540=1108.425,216.677,-68.923,-178.806,9.573,149.561
C01541=1108.421,216.925,-68.949,-178.804,9.576,149.561
C01542=1108.416,217.175,-68.976,-178.801,9.579,149.561
C01543=1108.412,217.423,-69.002,-178.799,9.583,149.561
C01544=1108.407,217.672,-69.028,-178.797,9.585,149.561
C01545=1108.403,217.920,-69.055,-178.795,9.588,149.561
C01546=1108.398,218.169,-69.081,-178.792,9.591,149.561
C01547=1108.394,218.417,-69.108,-178.790,9.595,149.562
C01548=1108.390,218.665,-69.134,-178.787,9.598,149.562
C01549=1108.385,218.915,-69.161,-178.786,9.600,149.562
C01550=1108.382,219.163,-69.187,-178.783,9.603,149.562
C01551=1108.377,219.411,-69.214,-178.781,9.606,149.562
C01552=1108.373,219.660,-69.240,-178.778,9.610,149.562
C01553=1108.368,219.909,-69.267,-178.776,9.613,149.562
C01554=1108.364,220.157,-69.293,-178.773,9.616,149.562
C01555=1108.359,220.406,-69.320,-178.771,9.618,149.562
C01556=1108.355,220.654,-69.346,-178.769,9.622,149.562
C01557=1108.351,220.903,-69.373,-178.766,9.625,149.562
C01558=1108.346,221.151,-69.400,-178.764,9.628,149.563
C01559=1108.342,221.400,-69.426,-178.762,9.631,149.563
C01560=1108.337,221.648,-69.453,-178.759,9.634,149.563
C01561=1108.333,221.897,-69.480,-178.757,9.637,149.563
C01562=1108.328,222.145,-69.507,-178.755,9.640,149.563
C01563=1108.325,222.393,-69.533,-178.752,9.643,149.563
C01564=1108.320,222.643,-69.560,-178.750,9.646,149.563
C01565=1108.316,222.892,-69.587,-178.748,9.649,149.563
C01566=1108.312,223.140,-69.613,-178.745,9.653,149.563
C01567=1108.307,223.388,-69.640,-178.743,9.656,149.563
C01568=1108.302,223.637,-69.667,-178.740,9.659,149.564
C01569=1108.298,223.885,-69.694,-178.738,9.661,149.564
C01570=1108.294,224.133,-69.721,-178.736,9.664,149.564
C01571=1108.289,224.382,-69.748,-178.733,9.667,149.564
C01572=1108.285,224.630,-69.775,-178.731,9.670,149.564
C01573=1108.280,224.879,-69.801,-178.728,9.674,149.564
C01574=1108.276,225.128,-69.828,-178.726,9.677,149.564
C01575=1108.272,225.377,-69.855,-178.723,9.680,149.564
C01576=1108.268,225.625,-69.882,-178.721,9.683,149.564
C01577=1108.263,225.874,-69.909,-178.719,9.685,149.564
C01578=1108.259,226.122,-69.935,-178.716,9.688,149.564
C01579=1108.254,226.370,-69.962,-178.713,9.691,149.564
C01580=1108.250,226.619,-69.989,-178.711,9.694,149.564
C01581=1108.246,226.868,-70.017,-178.708,9.697,149.564
C01582=1108.242,227.115,-70.044,-178.706,9.700,149.564
C01583=1108.237,227.328,-70.067,-178.704,9.703,149.564
C01584=1108.234,227.541,-70.090,-178.702,9.705,149.564
C01585=1108.231,227.754,-70.113,-178.699,9.708,149.564
C01586=1108.227,227.967,-70.136,-178.697,9.710,149.564
C01587=1108.223,228.179,-70.160,-178.695,9.713,149.564
C01588=1108.219,228.393,-70.183,-178.693,9.716,149.564
C01589=1108.216,228.605,-70.206,-178.690,9.718,149.564
C01590=1108.212,228.818,-70.229,-178.688,9.720,149.564
C01591=1108.207,229.067,-70.257,-178.686,9.723,149.564
C01592=1108.203,229.315,-70.284,-178.683,9.726,149.564
C01593=1108.198,229.564,-70.311,-178.680,9.729,149.564
C01594=1108.195,229.811,-70.338,-178.678,9.732,149.564
C01595=1108.190,230.060,-70.365,-178.675,9.735,149.564
C01596=1108.186,230.309,-70.392,-178.673,9.737,149.564
C01597=1108.181,230.557,-70.419,-178.670,9.740,149.564
C01598=1108.177,230.806,-70.446,-178.668,9.743,149.564
C01599=1108.172,231.054,-70.474,-178.665,9.746,149.564
C01600=1108.168,231.303,-70.502,-178.662,9.749,149.564
C01601=1108.163,231.552,-70.529,-178.660,9.751,149.564
C01602=1108.160,231.799,-70.556,-178.657,9.754,149.564
C01603=1108.156,232.048,-70.583,-178.654,9.757,149.564
C01604=1108.151,232.297,-70.610,-178.651,9.759,149.564
C01605=1108.147,232.545,-70.638,-178.649,9.762,149.564
C01606=1108.142,232.793,-70.665,-178.646,9.764,149.564
C01607=1108.138,233.042,-70.693,-178.644,9.767,149.564
C01608=1108.134,233.290,-70.720,-178.641,9.770,149.564
C01609=1108.129,233.539,-70.748,-178.638,9.773,149.564
C01610=1108.125,233.788,-70.775,-178.636,9.775,149.564
C01611=1108.121,234.036,-70.803,-178.633,9.778,149.563
C01612=1108.116,234.284,-70.830,-178.630,9.781,149.563
C01613=1108.112,234.533,-70.858,-178.627,9.784,149.563
C01614=1108.108,234.781,-70.885,-178.625,9.786,149.563
C01615=1108.103,235.029,-70.913,-178.622,9.789,149.563
C01616=1108.099,235.278,-70.940,-178.620,9.791,149.563
C01617=1108.095,235.526,-70.968,-178.617,9.793,149.563
C01618=1108.090,235.775,-70.995,-178.614,9.796,149.563
C01619=1108.086,236.023,-71.023,-178.611,9.799,149.563
C01620=1108.082,236.272,-71.050,-178.609,9.801,149.563
C01621=1108.077,236.520,-71.078,-178.607,9.804,149.563
C01622=1108.073,236.769,-71.105,-178.604,9.807,149.563
C01623=1108.069,237.017,-71.133,-178.601,9.810,149.562
C01624=1108.064,237.265,-71.160,-178.599,9.812,149.563
C01625=1108.060,237.514,-71.189,-178.596,9.815,149.562
C01626=1108.056,237.762,-71.217,-178.593,9.817,149.562
C01627=1108.051,238.011,-71.244,-178.591,9.819,149.562
C01628=1108.047,238.259,-71.272,-178.588,9.822,149.562
C01629=1108.043,238.507,-71.300,-178.585,9.825,149.562
C01630=1108.039,238.756,-71.327,-178.583,9.827,149.562
C01631=1108.034,239.004,-71.355,-178.580,9.830,149.562
C01632=1108.031,239.253,-71.383,-178.577,9.833,149.562
C01633=1108.025,239.501,-71.411,-178.575,9.835,149.562
C01634=1108.021,239.749,-71.439,-178.572,9.838,149.562
C01635=1108.017,239.998,-71.467,-178.569,9.841,149.562
C01636=1108.012,240.246,-71.494,-178.567,9.843,149.561
C01637=1108.009,240.495,-71.522,-178.564,9.846,149.561
C01638=1108.004,240.743,-71.550,-178.561,9.848,149.561
C01639=1108.000,240.956,-71.574,-178.559,9.850,149.561
C01640=1107.996,241.169,-71.598,-178.557,9.853,149.561
C01641=1107.993,241.382,-71.622,-178.555,9.855,149.561
C01642=1107.989,241.594,-71.646,-178.552,9.857,149.561
C01643=1107.986,241.806,-71.670,-178.550,9.860,149.561
C01644=1107.982,242.019,-71.693,-178.548,9.862,149.561
C01645=1107.979,242.232,-71.718,-178.546,9.864,149.561
C01646=1107.975,242.445,-71.741,-178.543,9.866,149.561
C01647=1107.970,242.693,-71.770,-178.541,9.869,149.561
C01648=1107.966,242.942,-71.798,-178.539,9.871,149.561
C01649=1107.962,243.189,-71.825,-178.536,9.874,149.561
C01650=1107.958,243.438,-71.854,-178.533,9.877,149.561
C01651=1107.953,243.686,-71.882,-178.530,9.880,149.561
C01652=1107.949,243.935,-71.910,-178.528,9.882,149.561
C01653=1107.945,244.183,-71.937,-178.525,9.885,149.561
C01654=1107.940,244.432,-71.966,-178.523,9.888,149.561
C01655=1107.936,244.680,-71.994,-178.520,9.890,149.561
C01656=1107.932,244.929,-72.022,-178.518,9.893,149.561
C01657=1107.927,245.177,-72.050,-178.515,9.896,149.561
C01658=1107.923,245.425,-72.078,-178.513,9.899,149.561
C01659=1107.919,245.673,-72.106,-178.510,9.901,149.560
C01660=1107.914,245.922,-72.135,-178.508,9.904,149.561
C01661=1107.910,246.170,-72.163,-178.505,9.907,149.561
C01662=1107.905,246.419,-72.191,-178.502,9.910,149.561
C01663=1107.902,246.668,-72.220,-178.500,9.912,149.561
C01664=1107.898,246.915,-72.248,-178.498,9.915,149.561
C01665=1107.893,247.164,-72.277,-178.495,9.918,149.561
C01666=1107.889,247.412,-72.305,-178.492,9.921,149.561
C01667=1107.884,247.660,-72.333,-178.490,9.924,149.561
C01668=1107.880,247.908,-72.361,-178.487,9.927,149.561
C01669=1107.875,248.157,-72.390,-178.484,9.930,149.561
C01670=1107.872,248.406,-72.418,-178.481,9.933,149.561
C01671=1107.867,248.654,-72.446,-178.478,9.936,149.560
C01672=1107.863,248.902,-72.475,-178.476,9.939,149.561
C01673=1107.859,249.150,-72.503,-178.473,9.942,149.560
C01674=1107.854,249.399,-72.532,-178.470,9.944,149.560
C01675=1107.851,249.647,-72.560,-178.467,9.947,149.560
C01676=1107.846,249.895,-72.588,-178.464,9.950,149.560
C01677=1107.842,250.143,-72.617,-178.462,9.952,149.560
C01678=1107.838,250.392,-72.646,-178.459,9.955,149.560
C01679=1107.833,250.640,-72.674,-178.456,9.957,149.560
C01680=1107.829,250.889,-72.702,-178.453,9.960,149.559
C01681=1107.825,251.137,-72.732,-178.450,9.962,149.559
C01682=1107.820,251.385,-72.760,-178.447,9.964,149.559
C01683=1107.816,251.634,-72.788,-178.444,9.967,149.559
C01684=1107.812,251.882,-72.817,-178.441,9.970,149.559
C01685=1107.807,252.130,-72.845,-178.439,9.972,149.559
C01686=1107.803,252.379,-72.874,-178.436,9.974,149.559
C01687=1107.799,252.627,-72.903,-178.433,9.977,149.558
C01688=1107.794,252.875,-72.931,-178.430,9.979,149.558
C01689=1107.791,253.123,-72.960,-178.427,9.981,149.558
C01690=1107.786,253.372,-72.989,-178.424,9.984,149.558
C01691=1107.782,253.621,-73.017,-178.422,9.986,149.558
C01692=1107.778,253.868,-73.046,-178.419,9.989,149.558
C01693=1107.773,254.117,-73.075,-178.417,9.991,149.557
C01694=1107.770,254.365,-73.104,-178.414,9.994,149.557
C01695=1107.766,254.578,-73.129,-178.411,9.996,149.557
C01696=1107.762,254.790,-73.153,-178.409,9.998,149.557
C01697=1107.758,255.003,-73.178,-178.407,10.000,149.557
C01698=1107.755,255.215,-73.202,-178.404,10.003,149.557
C01699=1107.751,255.427,-73.227,-178.402,10.005,149.557
C01700=1107.747,255.640,-73.252,-178.400,10.007,149.557
C01701=1107.744,255.853,-73.277,-178.398,10.009,149.557
C01702=1107.740,256.066,-73.301,-178.395,10.011,149.557
C01703=1107.736,256.314,-73.331,-178.393,10.014,149.557
C01704=1107.731,256.562,-73.359,-178.390,10.017,149.557
C01705=1107.728,256.810,-73.388,-178.387,10.020,149.557
C01706=1107.723,257.058,-73.417,-178.385,10.022,149.556
C01707=1107.719,257.307,-73.446,-178.382,10.025,149.557
C01708=1107.714,257.555,-73.475,-178.379,10.027,149.556
C01709=1107.710,257.803,-73.503,-178.376,10.030,149.556
C01710=1107.706,258.052,-73.533,-178.374,10.033,149.556
C01711=1107.702,258.300,-73.562,-178.371,10.036,149.556
C01712=1107.698,258.549,-73.591,-178.369,10.038,149.556
C01713=1107.693,258.797,-73.620,-178.366,10.041,149.556
C01714=1107.689,259.044,-73.649,-178.363,10.044,149.556
C01715=1107.685,259.292,-73.678,-178.360,10.047,149.556
C01716=1107.681,259.541,-73.707,-178.357,10.049,149.556
C01717=1107.676,259.790,-73.736,-178.354,10.052,149.556
C01718=1107.672,260.038,-73.766,-178.352,10.054,149.556
C01719=1107.668,260.286,-73.795,-178.349,10.057,149.556
C01720=1107.664,260.534,-73.823,-178.347,10.060,149.556
C01721=1107.660,260.782,-73.853,-178.344,10.063,149.556
C01722=1107.655,261.031,-73.882,-178.341,10.066,149.556
C01723=1107.651,261.279,-73.911,-178.338,10.068,149.555
C01724=1107.647,261.527,-73.941,-178.335,10.070,149.555
C01725=1107.643,261.776,-73.970,-178.332,10.073,149.555
C01726=1107.638,262.024,-73.999,-178.330,10.076,149.555
C01727=1107.634,262.273,-74.029,-178.327,10.079,149.555
C01728=1107.629,262.520,-74.058,-178.324,10.081,149.555
C01729=1107.625,262.768,-74.087,-178.321,10.084,149.555
C01730=1107.621,263.017,-74.117,-178.318,10.086,149.555
C01731=1107.617,263.265,-74.146,-178.315,10.089,149.555
C01732=1107.613,263.513,-74.175,-178.313,10.092,149.554
C01733=1107.609,263.761,-74.205,-178.310,10.094,149.554
C01734=1107.604,264.010,-74.234,-178.307,10.097,149.554
C01735=1107.600,264.258,-74.264,-178.304,10.099,149.554
C01736=1107.596,264.506,-74.293,-178.301,10.102,149.554
C01737=1107.592,264.755,-74.323,-178.298,10.105,149.554
C01738=1107.588,265.003,-74.352,-178.296,10.107,149.554
C01739=1107.583,265.251,-74.382,-178.292,10.110,149.554
C01740=1107.579,265.499,-74.411,-178.290,10.112,149.553
C01741=1107.575,265.748,-74.441,-178.287,10.115,149.553
C01742=1107.570,265.995,-74.470,-178.284,10.117,149.553
C01743=1107.566,266.243,-74.499,-178.281,10.120,149.553
C01744=1107.562,266.492,-74.529,-178.279,10.122,149.553
C01745=1107.558,266.740,-74.558,-178.276,10.125,149.553
C01746=1107.554,266.988,-74.587,-178.273,10.128,149.553
C01747=1107.550,267.236,-74.618,-178.270,10.130,149.553
C01748=1107.545,267.484,-74.647,-178.267,10.133,149.553
C01749=1107.541,267.732,-74.677,-178.265,10.135,149.552
C01750=1107.536,267.981,-74.707,-178.261,10.137,149.552
C01751=1107.532,268.310,-74.746,-178.258,10.141,149.552
C01752=1107.526,268.639,-74.785,-178.254,10.145,149.552
C01753=1107.520,268.968,-74.825,-178.250,10.148,149.552
C01754=1107.515,269.296,-74.864,-178.247,10.151,149.552
C01755=1107.511,269.544,-74.894,-178.244,10.154,149.552
C01756=1107.507,269.793,-74.923,-178.241,10.157,149.551
C01757=1107.502,270.041,-74.953,-178.238,10.160,149.551
C01758=1107.498,270.289,-74.983,-178.235,10.162,149.551
C01759=1107.494,270.537,-75.013,-178.233,10.164,149.551
C01760=1107.489,270.785,-75.042,-178.230,10.167,149.551
C01761=1107.485,271.033,-75.073,-178.227,10.170,149.551
C01762=1107.481,271.282,-75.103,-178.223,10.172,149.551
C01763=1107.477,271.531,-75.132,-178.220,10.175,149.551
C01764=1107.473,271.778,-75.163,-178.218,10.178,149.550
C01765=1107.469,272.027,-75.192,-178.215,10.180,149.550
C01766=1107.464,272.274,-75.223,-178.212,10.182,149.550
C01767=1107.460,272.523,-75.252,-178.209,10.185,149.550
C01768=1107.456,272.770,-75.282,-178.206,10.188,149.550
C01769=1107.452,273.019,-75.312,-178.203,10.191,149.550
C01770=1107.447,273.267,-75.342,-178.201,10.194,149.550
C01771=1107.443,273.515,-75.372,-178.198,10.196,149.550
C01772=1107.440,273.764,-75.402,-178.195,10.198,149.550
C01773=1107.435,274.012,-75.433,-178.192,10.201,149.550
C01774=1107.431,274.260,-75.462,-178.189,10.204,149.549
C01775=1107.427,274.508,-75.492,-178.186,10.207,149.549
C01776=1107.422,274.756,-75.523,-178.184,10.209,149.549
C01777=1107.418,275.004,-75.553,-178.181,10.211,149.549
C01778=1107.415,275.252,-75.583,-178.178,10.214,149.549
C01779=1107.410,275.501,-75.613,-178.175,10.216,149.549
C01780=1107.406,275.749,-75.643,-178.172,10.219,149.549
C01781=1107.402,275.996,-75.673,-178.169,10.222,149.549
C01782=1107.397,276.245,-75.703,-178.166,10.225,149.548
C01783=1107.393,276.492,-75.734,-178.163,10.228,149.548
C01784=1107.389,276.742,-75.764,-178.161,10.230,149.548
C01785=1107.385,276.989,-75.794,-178.158,10.232,149.548
C01786=1107.381,277.237,-75.825,-178.155,10.235,149.548
C01787=1107.377,277.485,-75.855,-178.152,10.237,149.548
C01788=1107.373,277.734,-75.885,-178.149,10.240,149.548
C01789=1107.369,277.982,-75.916,-178.146,10.243,149.548
C01790=1107.365,278.230,-75.946,-178.144,10.245,149.547
C01791=1107.122,267.658,-74.726,-178.264,10.135,149.552
C01792=1107.127,267.410,-74.696,-178.267,10.133,149.552
C01793=1107.131,267.161,-74.667,-178.270,10.130,149.552
C01794=1107.135,266.913,-74.637,-178.272,10.127,149.553
C01795=1107.139,266.665,-74.608,-178.275,10.124,149.553
C01796=1107.143,266.417,-74.577,-178.278,10.122,149.553
C01797=1107.147,266.169,-74.548,-178.281,10.120,149.553
C01798=1107.152,265.921,-74.519,-178.284,10.117,149.553
C01799=1107.156,265.673,-74.489,-178.287,10.115,149.553
C01800=1107.161,265.425,-74.460,-178.290,10.112,149.553
C01801=1107.165,265.176,-74.431,-178.292,10.110,149.554
C01802=1107.169,264.928,-74.401,-178.295,10.107,149.554
C01803=1107.173,264.680,-74.372,-178.298,10.104,149.554
C01804=1107.177,264.432,-74.342,-178.301,10.101,149.554
C01805=1107.181,264.183,-74.313,-178.304,10.099,149.554
C01806=1107.186,263.935,-74.283,-178.307,10.097,149.554
C01807=1107.190,263.687,-74.254,-178.310,10.094,149.554
C01808=1107.194,263.439,-74.224,-178.313,10.092,149.554
C01809=1107.198,263.190,-74.195,-178.315,10.089,149.555
C01810=1107.202,262.942,-74.165,-178.318,10.087,149.555
C01811=1107.207,262.694,-74.136,-178.321,10.084,149.555
C01812=1107.211,262.445,-74.107,-178.324,10.081,149.555
C01813=1107.216,262.197,-74.078,-178.327,10.079,149.555
C01814=1107.220,261.949,-74.049,-178.330,10.076,149.555
C01815=1107.224,261.701,-74.019,-178.332,10.074,149.555
C01816=1107.228,261.453,-73.990,-178.335,10.071,149.555
C01817=1107.233,261.204,-73.960,-178.337,10.068,149.555
C01818=1107.237,260.956,-73.931,-178.340,10.065,149.555
C01819=1107.241,260.708,-73.901,-178.343,10.062,149.555
C01820=1107.245,260.459,-73.873,-178.346,10.060,149.556
C01821=1107.249,260.212,-73.844,-178.348,10.058,149.556
C01822=1107.254,259.963,-73.815,-178.351,10.055,149.556
C01823=1107.258,259.715,-73.785,-178.354,10.052,149.556
C01824=1107.262,259.466,-73.757,-178.357,10.049,149.556
C01825=1107.267,259.218,-73.727,-178.360,10.046,149.556
C01826=1107.270,258.970,-73.698,-178.363,10.044,149.556
C01827=1107.275,258.722,-73.669,-178.365,10.042,149.556
